(* CoDeSys 2.3.9.62 project: MM000-P9020-00-A.pro *)
(* Author: JvL *)
(* Libraries: ifm_CR0451\ifm_CR0451_Init_V030000.lib 23.10.20 12:28:47, ifm_CR0451\ifm_CR0451_V030002.lib 22.3.17 09:59:30, ifm_RAWCan\ifm_RAWCan_NT_V020004.lib 1.10.19 08:10:40, ifm_CANopen\ifm_CANopen_NT_V020004.lib 1.10.19 08:10:40, ifm_CANopen\ifm_NetVarLib_NT_V020004.lib 1.10.19 08:10:40, ifm_CANopen\3S_CANopenManager.lib 23.10.20 12:28:45, ifm_CANopen\3S_CanDrv.lib 23.10.20 12:28:45, Util.lib 23.10.20 12:25:49, ifm_PDMsmart_util_V010007.lib 23.10.20 12:28:45, Iecsfc.lib 2.6.14 11:37:46, 3S_CANOPENNETVAR.LIB 23.10.20 12:28:45, standard.lib 4.10.05 12:14:46, SysLibVisuBasicDisplay.lib 22.3.17 09:59:30, SysLibTargetVisu.lib 5.4.04 14:31:00, SysLibCallback.lib 26.9.08 18:43:52, ifm_CR0451_callback_visu.lib 23.10.20 12:28:47, SysLibStr.lib 13.6.03 16:49:00 *)

(* PLC configuration (modules and I/O channels)
CR0451 Configuration V03 [Root] node -1, in %IB0 out %QB0
  Configuration [LocalConfiguration] node 0, in %IB0 out %QB0 {IFM_PARAM_WORD_TIME = 10}
  Input/Output [LocalInputOutput] node 1, in %IB0 out %QB0
    Display Keys [LocalKeys] node 0, in %IB0 out %QB0
      KEY_F1 AT %IB0 [ChInputBool] F1 Key
      KEY_F2 AT %IB1 [ChInputBool] F2 Key
      KEY_F3 AT %IB2 [ChInputBool] F3 Key
      KEY_F4 AT %IB3 [ChInputBool] F4 Key
      KEY_UP AT %IB4 [ChInputBool] Up Key
      KEY_DOWN AT %IB5 [ChInputBool] Down Key
      KEY_LEFT AT %IB6 [ChInputBool] Left Key
      KEY_RIGHT AT %IB7 [ChInputBool] Right Key
      KEY_OK AT %IB8 [ChInputBool] Ok Key
    Virtual Raising Keys [VirtualRaisingKeys] node 1, in %IB9 out %QB0
      RT_F1 AT %IB9 [ChInputBool] Rising Edge F1 Key
      RT_F2 AT %IB10 [ChInputBool] Rising Edge F2 Key
      RT_F3 AT %IB11 [ChInputBool] Rising Edge F3 Key
      RT_F4 AT %IB12 [ChInputBool] Rising Edge F4 Key
      RT_UP AT %IB13 [ChInputBool] Rising Edge Up Key
      RT_DOWN AT %IB14 [ChInputBool] Rising Edge Down Key
      RT_LEFT AT %IB15 [ChInputBool] Rising Edge Left Key
      RT_RIGHT AT %IB16 [ChInputBool] Rising Edge Right Key
      RT_OK AT %IB17 [ChInputBool] Rising Edge Ok Key
    Virtual Falling Keys [VirtualFallingKeys] node 2, in %IB18 out %QB0
      FT_F1 AT %IB18 [ChInputBool] Falling Edge F1 Key
      FT_F2 AT %IB19 [ChInputBool] Falling Edge F2 Key
      FT_F3 AT %IB20 [ChInputBool] Falling Edge F3 Key
      FT_F4 AT %IB21 [ChInputBool] Falling Edge F4 Key
      FT_UP AT %IB22 [ChInputBool] Falling Edge Up Key
      FT_DOWN AT %IB23 [ChInputBool] Falling Edge Down Key
      FT_LEFT AT %IB24 [ChInputBool] Falling Edge Left Key
      FT_RIGHT AT %IB25 [ChInputBool] Falling Edge Right Key
      FT_OK AT %IB26 [ChInputBool] Falling Edge Ok Key
    Key Events [KeyEvents] node 3, in %IB27 out %QB0
      KEY_CHANGED AT %IB27 [ChInputBool] Event: Key Changed
      KEY_PRESSED AT %IB28 [ChInputBool] Event: Key is pressed
    System Inputs [LocalSystemInputs] node 4, in %IB29 out %QB0
      SUPPLY_VOLTAGE_VBBS AT %IW15 [ChInputWord] Supply voltage VBBS
      SUPPLY_VOLTAGE_VU AT %IW16 [ChInputWord] Supply voltage VU
      TEMPERATURE AT %IW17 [ChInputInt] Temperature
    Backlight Control [LocalBacklightControl] node 5, in %IB36 out %QB0
      SCREEN_BACKLIGHT_CTRL AT %QB0 [ChOutputByte] Screen Backlight (0 - 100%)
      KEY_BACKLIGHT_CTRL AT %QB1 [ChOutputByte] Key Backlight (0 - 100%)
  CAN Communication [LocalCANCom] node 2, in %IB36 out %QB2
    Interface CAN 1 [CAN_BUS] node 0, in %IB36 out %QB2 {STACK_DWORD_S = 0}
      CANopen Interface [CAN_OPEN] node 0, in %IB36 out %QB2
      J1939 Interface [CAN_J1939] node 1, in %IB36 out %QB2
*)

(* Global variable list: CanOpen implicit Variables *)
VAR_GLOBAL CONSTANT
	MAX_CTRLINDEX : INT := -1;
END_VAR

(* Global variable list: Global_Variables *)
VAR_GLOBAL
	alarm: BOOL;
	editMode: BOOL;
	brakesAlarm: BOOL;
	overloadWarningBlink: BOOL;
	sensorFailureBlink: BOOL;
	overspeedAlarmBlink: BOOL;
	cr0451VersionNo: STRING;
	prefix: STRING;
END_VAR

VAR_GLOBAL RETAIN
	bandLimit: BYTE;
	wcbLimit: BYTE;
END_VAR

(* Global variable list: Networkmanagement implicit Variables CAN *)
VAR_GLOBAL CONSTANT
	USE_NWVARS_CAN : BOOL := TRUE;
	MAX_NetVarItems_CAN	: INT := 23;
	MAX_NetVarPDO_Rx_CAN	: INT := 6;
	MAX_NetVarPDO_Tx_CAN	: INT := 0;
	MAX_NetVarOD_CAN		: INT := 0;
END_VAR
VAR_GLOBAL
	pNetVarItems_CAN		: ARRAY[0..MAX_NetVarItems_CAN] OF NetVarDataItem_CAN;
	pNetVarPDO_Rx_CAN		: ARRAY[0..MAX_NetVarPDO_Rx_CAN] OF NetVarPDO_Rx_CAN;
	pNetVarPDO_Tx_CAN		: ARRAY[0..MAX_NetVarPDO_Tx_CAN] OF NetVarPDO_Tx_CAN;
	pNetVarOD_CAN			: ARRAY[0..MAX_NetVarOD_CAN] OF NetVarOD_CAN;
END_VAR

(* Global variable list: PDM_PLC_COMUNICATION2 *)
VAR_GLOBAL

	(*
	 System variables for basic comunication. CANopen TX/RX PDO1, PDO2, PDO3 and PDO4
	or CANLayer2 TX/RX COB1, COB2, COB3 and COB4
	*)


(************************************From PDM to PLC**********************************************************)

	PRESENT_PAGE:WORD;					(*Preset page number from PDM to PLC*)
	PRESENT_MESSAGE:BYTE;					(*Preset message number from PDM to PLC*)
	PRESENT_MESSAGE_GROUP:BYTE;		(*Preset message group number from PDM to PLC*)
	F_KEYS:BYTE;								(*Funtion keys F1 to F8 from PDM to PLC*)
	C_KEYS:BYTE;								(*Control keys from PDM to PLC*)
	PRESENT_LEDVALUE_MAX:BYTE;			(*Preset LED valus max from PDM to PLC*)
	PRESENT_LEDVALUE_NIGHT:BYTE;		(*Preset LED value night from PDM to PLC*)

	PRESENT_BACKLIGHT:BYTE;				(*Preset backlight value from PDM to PLC*)
	HANDLE:WORD;								(*Handle for input value to PLC*)
	INPUT_VALUE:DWORD;						(*Input value to PLC*)
	LENGHT:BYTE;								(*Length for input value*)

	F_KEYS2:				BYTE;					(*Funtion keys F9 to F16 from PDM to PLC*)
	ToPlcPdo3ReserveByte1:BYTE;					(*Reserve PDO*)
	ToPlcPdo3ReserveByte2:BYTE;					(*Reserve PDO*)
	ToPlcPdo3ReserveByte3:BYTE;					(*Reserve PDO*)
	ToPlcPdo3ReserveByte4:BYTE;					(*Reserve PDO*)
	ToPlcPdo3ReserveByte5:BYTE;					(*Reserve PDO*)
	ToPlcPdo3ReserveByte6:BYTE;					(*Reserve PDO*)
	ToPlcPdo3ReserveByte7:BYTE;					(*Reserve PDO*)

	ToPlcPdo4ReserveByte0:BYTE;					(*Reserve PDO*)
	ToPlcPdo4ReserveByte1:BYTE;					(*Reserve PDO*)
	ToPlcPdo4ReserveByte2:BYTE;					(*Reserve PDO*)
	ToPlcPdo4ReserveByte3:BYTE;					(*Reserve PDO*)
	ToPlcPdo4ReserveByte4:BYTE;					(*Reserve PDO*)
	ToPlcPdo4ReserveByte5:BYTE;					(*Reserve PDO*)
	ToPlcPdo4ReserveByte6:BYTE;					(*Reserve PDO*)
	ToPlcPdo4ReserveByte7:BYTE;					(*Reserve PDO*)

(*^^^^^^^^^^^^^^^^^^^^^^^^^^^^^^^^^^^^^^^^^^^^^^^^^^^^^^^^^^^^^^^^^^^^^^^^^^^^^^^^^^^^^^^^^^^^^^^^^^^^^^^^^^^^^^^^^^^^^^^^^^^^^^^^^^^^^^^^^^*)

(*********************************************From PLC to PDM****************************************************************************)

	DESIRED_PAGE:WORD;						(*Desired page number from PLC to PDM*)
	DESIRED_MESSAGE:BYTE;					(*Desired message number from PLC to PDM*)
	DESIRED_MESSAGE_GROUP:BYTE;		(*Desired message group number from PLC to PDM*)
	LED_F_KEYS:BYTE;							(*LED Funtion keys F1 to F8 from PLC to PDM*)
	LED_C_KEYS:BYTE;							(*LED Control keys from PLC to PDM*)
	DESIRED_LEDVALUE_MAX:BYTE;			(*Desired LED valus max from PLC to PDM*)
	DESIRED_LEDVALUE_NIGHT:BYTE;		(*Desired LED value night from PLC to PDM*)

	DESIRED_BACKLIGHT:BYTE;				(*Desired backlight value from PLC to PDM*)
	HANDLE_BACK:WORD;						(*Handle for input value, write back from PLC*)
	INPUT_VALUE_BACK:DWORD;				(*Input value, write back from PLC*)
	LENGHT_BACK:BYTE;						(*Length for input value, write back from PLC*)

	LED_F_KEYS2		:BYTE;					(*LED Funtion keys F9 to F16 from PLC to PDM*)
	ToPdmPdo3ReserveByte1:BYTE;					(*Reserve PDO*)
	ToPdmPdo3ReserveByte2:BYTE;					(*Reserve PDO*)
	ToPdmPdo3ReserveByte3:BYTE;					(*Reserve PDO*)
	ToPdmPdo3ReserveByte4:BYTE;					(*Reserve PDO*)
	ToPdmPdo3ReserveByte5:BYTE;					(*Reserve PDO*)
	ToPdmPdo3ReserveByte6:BYTE;					(*Reserve PDO*)
	ToPdmPdo3ReserveByte7:BYTE;					(*Reserve PDO*)

	ToPdmPdo4ReserveByte0:BYTE;					(*Reserve PDO*)
	ToPdmPdo4ReserveByte1:BYTE;					(*Reserve PDO*)
	ToPdmPdo4ReserveByte2:BYTE;					(*Reserve PDO*)
	ToPdmPdo4ReserveByte3:BYTE;					(*Reserve PDO*)
	ToPdmPdo4ReserveByte4:BYTE;					(*Reserve PDO*)
	ToPdmPdo4ReserveByte5:BYTE;					(*Reserve PDO*)
	ToPdmPdo4ReserveByte6:BYTE;					(*Reserve PDO*)
	ToPdmPdo4ReserveByte7:BYTE;					(*Reserve PDO*)

(*^^^^^^^^^^^^^^^^^^^^^^^^^^^^^^^^^^^^^^^^^^^^^^^^^^^^^^^^^^^^^^^^^^^^^^^^^^^^^^^^^^^^^^^^^^^^^^^^^^^^^^^^^^^^^^^^^^^^^^^^^^^^^^^^^^^^^^^^^^*)

END_VAR

(* Global variable list: SOFTKEYFIELD *)
VAR_GLOBAL

	(*Variables Input and for text attribute*)
	InputModeDt: BOOL;
	TextColor:DWORD:=16#FFFFFF;
	TextSize:BYTE:=12;

	(*Variables to hide and show the key fields*)
	Hidden_F1:BOOL;
	Hidden_F2:BOOL;
	Hidden_F3:BOOL;
	Hidden_F4:BOOL;
	Hidden_F5:BOOL;
	Hidden_F6:BOOL;
	Hidden_F7:BOOL;
	Hidden_F8:BOOL;
	Hidden_F9:BOOL;
	Hidden_Ctrl:BOOL;
	Hidden_Up:BOOL;
	Hidden_Down:BOOL;
	Hidden_Left:BOOL;
	Hidden_Right:BOOL;
	Hidden_Ok:BOOL;
	Hidden_HeadLine:BOOL;

	(*
	String variables for softkeys.
	With string size 14 it ist possible to show two lines with 6 characters.
	Two character are use for CR/LF Ee.g.ROW_11 $R$NROW_22
	*)
	TXT_F1:STRING[20];
	TXT_F2:STRING[20];
	TXT_F3:STRING[20];
	TXT_F4:STRING[20];
	TXT_F5:STRING[20];
	TXT_F6:STRING[20];
	TXT_F7: STRING[20];
	TXT_F8: STRING[20];
	TXT_F9: STRING[20];
	TXT_Ctrl: STRING[20];
	TXT_HeadLine :STRING[30];

END_VAR

(* Global variable list: SoftKeys2Global *)
VAR_GLOBAL
(*Soft key's as R_TRIG*)
	SoftKey_F1: BOOL;
	SoftKey_F2: BOOL;
	SoftKey_F3: BOOL;
	SoftKey_F4: BOOL;
	SoftKey_F5: BOOL;
	SoftKey_F6: BOOL;
	SoftKey_F7: BOOL;
	SoftKey_F8: BOOL;
	SoftKey_F9: BOOL;
	SoftKey_F10: BOOL;
	SoftKey_Up: BOOL;
	SoftKey_Esc: BOOL;
	SoftKey_Ok: BOOL;
	SoftKey_Left: BOOL;
	SoftKey_Down: BOOL;
	SoftKey_Right: BOOL;
(*Soft key's as switch*)
	SoftKey2_F1: BOOL;
	SoftKey2_F2: BOOL;
	SoftKey2_F3: BOOL;
	SoftKey2_F4: BOOL;
	SoftKey2_F5: BOOL;
	SoftKey2_F6: BOOL;
	SoftKey2_F7: BOOL;
	SoftKey2_F8: BOOL;
	SoftKey2_F9: BOOL;
	SoftKey2_F10: BOOL;
	SoftKey2_Up: BOOL;
	SoftKey2_Esc: BOOL;
	SoftKey2_Ok: BOOL;
	SoftKey2_Left: BOOL;
	SoftKey2_Down: BOOL;
	SoftKey2_Right: BOOL;
	InputMode:BOOL;

END_VAR

(* POU PLC_PRG, FBD *)
PROGRAM PLC_PRG
(*******************************************************************************************************************

			Template for CR0451 V03 - CAN layer 2 (2014)
			--------------------------------------------

	Wir möchten an dieser Stelle ausdrücklich darauf hinweisen, dass die eingestellten Beispiele
	nicht ungeprüft industriell eingesetzt werden dürfen. Das heißt, dass wir für die Funktionalität
	insbesondere an Maschinen und Anlagen keinerlei Garantie übernehmen. Das Beispiel ist
	ausschließlich für Testzwecke bei der Entwicklung neuer Maschinen und Anlagen vorgesehen
	und wurde dafür in Abstimmung mit Ihnen konstruiert und hergestellt. Insoweit handelt es sich
	nicht um ein (Software-) Produkt, das von europäischen Richtlinien erfasst wird. Die Konformität
	mit einschlägigen Richtlinien und Normen zur Erfüllung der gesetzlichen Anforderungen für das
	Inverkehrbringen werden erst mit der Verifizierung und Validierung im Rahmen Ihrer Entwicklung
	festgestellt. Ein Bereitstellen auf dem Markt zur Verwendung durch Endnutzer darf bis zu diesem
	Zeitpunkt nicht stattfinden. 
 
 	We would like to expressly point out that the examples made available must not be used for industrial
	purposes without checking. We assume no guarantee whatsoever for their functionality, particularly
	regarding machines and plants. The example is only intended for testing during the development of
	new machines and plants and has been designed and manufactured for this purpose in coordination
	with you.  Consequently, it is not a (software) product subject to European directives. Compliance with
	relevant directives and standards to meet legal requirements regarding the placing on the market will
	only be determined during the verification and validation in the context of your development. Until then,
	it must not be put onto the market for use by end users.

*******************************************************************************************************************)

VAR

	init_1: BOOL := TRUE;
	CycleTime:DWORD;
	MaxCycleTime:DWORD;
	ResetMax:BOOL;

	Start_time: TIME;


	fbBlink02: BLINK;
END_VAR
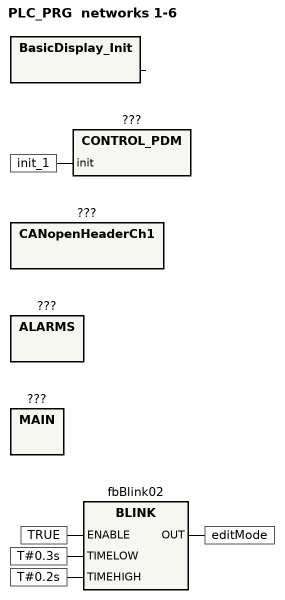
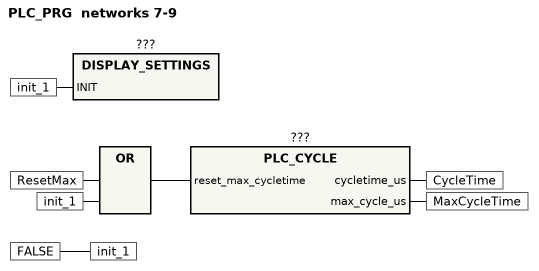
_FBD_ (* Function Block Diagram *)
NETWORK 1
	BasicDisplay_Init()
NETWORK 2
	???:CONTROL_PDM(init: init_1)
NETWORK 3
	???:CANopenHeaderCh1()
NETWORK 4
	???:ALARMS()
NETWORK 5
	???:MAIN()
NETWORK 6
	fbBlink02:BLINK(ENABLE: TRUE, TIMELOW: T#0.3s, TIMEHIGH: T#0.2s) => editMode
NETWORK 7
	???:DISPLAY_SETTINGS(INIT: init_1)
NETWORK 8
	???:PLC_CYCLE(reset_max_cycletime: OR(ResetMax, init_1), max_cycle_us => MaxCycleTime) => CycleTime
NETWORK 9 (* second last line *)
	FALSE => init_1
_END_FBD_
(* the same logic as Structured Text *)
(* Network 1 *)
BasicDisplay_Init();
(* Network 2: see the listing above *)
(* Network 3: see the listing above *)
(* Network 4: see the listing above *)
(* Network 5: see the listing above *)
(* Network 6 *)
fbBlink02(ENABLE := TRUE, TIMELOW := T#0.3s, TIMEHIGH := T#0.2s);
editMode := fbBlink02.OUT;
(* Network 7: see the listing above *)
(* Network 8: see the listing above *)
(* Network 9 *)
init_1 := FALSE;
END_PROGRAM

(* POU CONTROL_CR10xx/CONTROL_PDM, FBD *)
PROGRAM CONTROL_PDM
VAR

	PageIntern: WORD;


	ErrorCom: BOOL;
END_VAR
VAR_INPUT

	init: BOOL;

END_VAR
VAR_OUTPUT
END_VAR
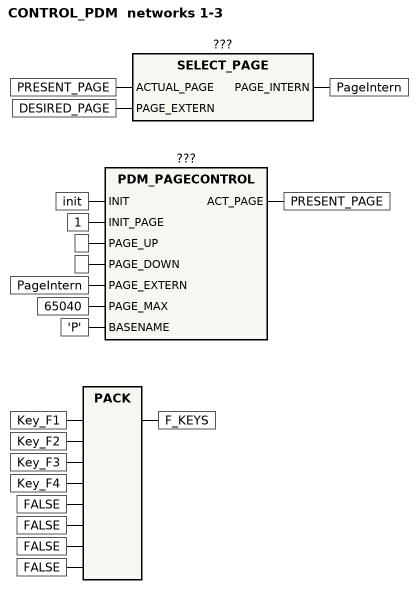
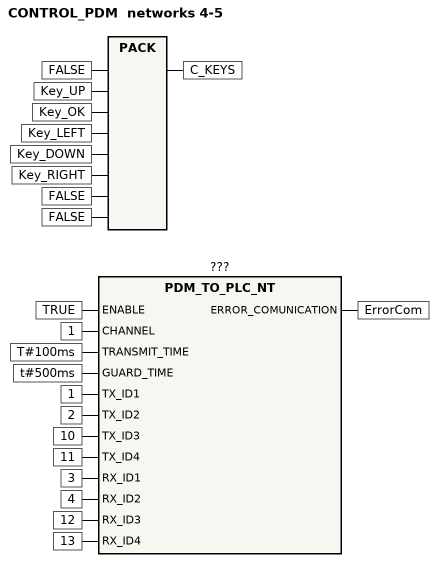
_FBD_ (* Function Block Diagram *)
NETWORK 1 (* This POU must located before PDM_PAGECONTROL, for timing reasons. Include here the program part to change the pages. *)
	???:SELECT_PAGE(ACTUAL_PAGE: PRESENT_PAGE, PAGE_EXTERN: DESIRED_PAGE) => PageIntern
NETWORK 2
	???:PDM_PAGECONTROL(INIT: init, INIT_PAGE: 1, PAGE_UP: , PAGE_DOWN: , PAGE_EXTERN: PageIntern, PAGE_MAX: 65040, BASENAME: 'P') => PRESENT_PAGE
NETWORK 3
	PACK(Key_F1, Key_F2, Key_F3, Key_F4, FALSE, FALSE, FALSE, FALSE) => F_KEYS
NETWORK 4
	PACK(FALSE, Key_UP, Key_OK, Key_LEFT, Key_DOWN, Key_RIGHT, FALSE, FALSE) => C_KEYS
NETWORK 5
	???:PDM_TO_PLC_NT(ENABLE: TRUE, CHANNEL: 1, TRANSMIT_TIME: T#100ms, GUARD_TIME: t#500ms, TX_ID1: 1, TX_ID2: 2, TX_ID3: 10, TX_ID4: 11, RX_ID1: 3, RX_ID2: 4, RX_ID3: 12, RX_ID4: 13) => ErrorCom
_END_FBD_
(* the same logic as Structured Text *)
(* Network 1: see the listing above *)
(* Network 2: see the listing above *)
(* Network 3 *)
F_KEYS := PACK(Key_F1, Key_F2, Key_F3, Key_F4, FALSE, FALSE, FALSE, FALSE);
(* Network 4 *)
C_KEYS := PACK(FALSE, Key_UP, Key_OK, Key_LEFT, Key_DOWN, Key_RIGHT, FALSE, FALSE);
(* Network 5: see the listing above *)
END_PROGRAM

(* POU CONTROL_CR10xx/SELECT_PAGE, ST *)
PROGRAM SELECT_PAGE
(*insert this POU in POU  CONTROL_PDM one line be for PDM_PAGECONTROL!!!!!!!!!!!!!!!!!*)
(*adapt the menue structure for your program in this POU*)
(*10.09.2010 vl FB enhanced by SoftKey2_F1 to SoftKey2_Right as switch*)

VAR_OUTPUT
	PAGE_INTERN: WORD;
END_VAR
VAR_INPUT
	ACTUAL_PAGE: WORD;
	PAGE_EXTERN:WORD;

END_VAR
VAR

	PageExternOld: WORD;

(*Virtual F-keys*)
	VirtualF1: BOOL;
	VirtualF2: BOOL;
	VirtualF3: BOOL;
	VirtualF4: BOOL;
	VirtualF5: BOOL;
	VirtualF6: BOOL;
	VirtualEsc: BOOL;
	VirtualUp: BOOL;
	VirtualOk: BOOL;
	VirtualLeft: BOOL;
	VirtualDown: BOOL;
	VirtualRight: BOOL;

	InputModeStep1: BOOL;
	InputPage: BOOL;
	InputMode:BOOL;
	TOF_InputMode: TOF;
	F_TRIG_InputMode: F_TRIG;

	F5: BOOL;
	InitMenu: BOOL;
	CountMenu: BYTE;
	MenuUp: BOOL;
	MenuDown: BOOL;
	MenuItem: BYTE;
	ItemOk: BOOL;

	Delay: TON;
END_VAR
(*Create virtual keys for menu's*)
	SELECT_MENU(
		Count:=CountMenu,
		Up:= MenuUp,
		Down:=MenuDown,
		MenuItem=>MenuItem );

	VirtualF1:=MenuItem=1 AND Key_Ok;
	VirtualF2:=MenuItem=2 AND Key_Ok;
	VirtualF3:=MenuItem=3 AND Key_Ok;
	VirtualF4:=MenuItem=4 AND Key_Ok;
	VirtualF5:=MenuItem=5 AND Key_Ok;
	VirtualF6:=MenuItem=6 AND Key_Ok;
(*^^^^^^^^^^^^^^^^^^^^^^^^^^^^^^^^^^^^^^^^^^^^^^^^^^^^^^^^^^^^^^^^^^^^^^^^^^^^^^^^^^^^^^^^^^*)

(*Use on following pages the real keys*)
	CASE ACTUAL_PAGE OF
		10:
				VirtualF1:= Key_F1;
				VirtualF2:= Key_F2;
				VirtualF3:= Key_F3;
		12:
				VirtualF1:= Key_F1;
				VirtualF2:= Key_F2;
				VirtualF4:= Key_F4;
		65020:
				VirtualF1:= Key_F1;
				VirtualF2:= Key_F2;
		65030:
				VirtualF1:= Key_F1;

	END_CASE;
(*^^^^^^^^^^^^^^^^^^^^^^^^^^^^^^^^^^^^^^^^^^^^^^^^^^^^^^^^^^^^^^^^^^^^^^^^^^^^^^^^^^^^^^^^^^*)

(*Create soft keys*)
	RT_SOFT_KEYS2(
		KEY_F1:=VirtualF1,
		KEY_F2:=VirtualF2,
		KEY_F3:=VirtualF3,
		KEY_F4:=VirtualF4,
		KEY_F5:=VirtualF5,
		KEY_F6:=VirtualF6,
		KEY_ESC:=Key_F4,
		KEY_UP:=KEY_UP,
		KEY_OK:=KEY_OK,
		KEY_LEFT:=KEY_LEFT,
		KEY_DOWN:=KEY_DOWN,
		KEY_RIGHT:=KEY_RIGHT );
(*^^^^^^^^^^^^^^^^^^^^^^^^^^^^^^^^^^^^^^^^^^^^^^^^^^^^^^^^^^^^^^^^^^^^^^^^^^^^^^^^^^^^^^^^^^*)

(*Set input mode for PDMsmart*)
	IF InputPage AND (SoftKey_LEFT OR SoftKey_RIGHT) THEN
		InputModeStep1:=TRUE;
	END_IF;
	IF SoftKey_ESC THEN
		InputModeStep1:=FALSE;
	END_IF;
	IF InputMode AND (SoftKey_ESC OR SoftKey_OK) THEN
		InputMode:=FALSE;
		InputModeStep1:=FALSE;
	END_IF;
	IF InputModeStep1 AND NOT InputMode AND SoftKey_OK THEN
		InputMode:=TRUE;
	END_IF;

(*^^^^^^^^^^^^^^^^^^^^^^^^^^^^^^^^^^^^^^^^^^^^^^^^^^^^^^^^^^^^^^^^^^^^^^^^^^^^^^^^^^^^^^^*)

(****PAGE from extern****************)
	IF PageExternOld<>PAGE_EXTERN THEN
		PageExternOld:=PAGE_EXTERN;
		PAGE_INTERN:=PAGE_EXTERN;
	END_IF;
(*^^^^^^^^^^^^^^^^^^^^^^^^^^^^^^^^^^^^^^^^^^^^^^^^^^^^^^^^^^^^^^^^*)

	CASE ACTUAL_PAGE OF
(********************Start page*******************************)

		1:	Delay(IN:= NOT(Delay.Q), PT:= T#3s);
			IF Delay.Q THEN
				PAGE_INTERN:= 10;
			END_IF
			InputPage:=FALSE;

			TXT_F1:='';
			TXT_F2:='';
			TXT_F3:='';
			TXT_F4:='';
			TXT_HeadLine:='';
			Hidden_F1:=TRUE;
			Hidden_F2:=TRUE;
			Hidden_F3:=TRUE;
			Hidden_F4:=TRUE;
			Hidden_Up:=TRUE;
			Hidden_Down:=TRUE;
			Hidden_Left:=TRUE;
			Hidden_Right:=TRUE;
			Hidden_Ok:=FALSE;
			Hidden_HeadLine:=FALSE;


(*^^^^^^^^^^^^^^^^^^^^^^^^^^^^^^^^^^^^^^^^^^^^^^^^^^^^^^^^^^^^^*)

(**************************Main page***********************************)
		10:
			Delay(IN:= NOT(Delay.Q), PT:= T#1s);
			IF Delay.Q THEN
				PAGE_INTERN:= 10;
			END_IF
			TXT_F1:='';
			TXT_F2:='';
			TXT_F3:='';
			TXT_F4:='';
			TXT_HeadLine:= '';
			Hidden_F1:=TRUE;
			Hidden_F2:=TRUE;
			Hidden_F3:=TRUE;
			Hidden_F4:=TRUE;
			Hidden_Up:=TRUE;
			Hidden_Down:=TRUE;
			Hidden_Left:=TRUE;
			Hidden_Right:=TRUE;
			Hidden_Ok:=TRUE;
			Hidden_HeadLine:=TRUE;

			IF SoftKey_F1 THEN
				PAGE_INTERN:= 16;
			END_IF
			IF SoftKey_F3 AND sensorFailure = FALSE THEN
				PAGE_INTERN:= 12;
				skylineActive:= TRUE;
			END_IF

			InputPage:=FALSE;

(********************************Input status page********************************************)
		11:
			TXT_F1:='';
			TXT_F2:='';
			TXT_F3:='';
			TXT_F4:= '';
			TXT_HeadLine:= 'INPUT STATUS';
			Hidden_F1:= TRUE;
			Hidden_F2:= TRUE;
			Hidden_F3:= TRUE;
			Hidden_F4:= TRUE;
			Hidden_Up:= TRUE;
			Hidden_Down:= TRUE;
			Hidden_Left:= TRUE;
			Hidden_Right:= TRUE;
			Hidden_Ok:= TRUE;
			Hidden_HeadLine:= FALSE;

			IF SoftKey_ESC THEN
				PAGE_INTERN:=16;
			END_IF;

			InputPage:=FALSE;

(********************************Working mode page********************************************)
		12:
			TXT_F1:='';
			TXT_F2:='';
			TXT_F3:='';
			TXT_F4:='';
			TXT_HeadLine:='';
			Hidden_F1:=TRUE;
			Hidden_F2:=TRUE;
			Hidden_F3:=TRUE;
			Hidden_F4:=TRUE;
			Hidden_Up:=TRUE;
			Hidden_Down:=TRUE;
			Hidden_Left:=TRUE;
			Hidden_Right:=TRUE;
			Hidden_Ok:=TRUE;
			Hidden_HeadLine:=FALSE;

			IF SoftKey_F1 THEN
				PAGE_INTERN:= 16;
			END_IF
			IF SoftKey_F2 THEN
				PAGE_INTERN:= 11;
			END_IF
			IF SoftKey_ESC OR sensorFailure = TRUE THEN
				PAGE_INTERN:= 10;
				skylineActive:= FALSE;
			END_IF;

			InputPage:=FALSE;

(********************************Alarm log page********************************************)
		13:
			TXT_F1:='';
			TXT_F2:='';
			TXT_F3:='';
			TXT_F4:='';
			TXT_HeadLine:='ALARMS LOG';
			Hidden_F1:=TRUE;
			Hidden_F2:=TRUE;
			Hidden_F3:=TRUE;
			Hidden_F4:=TRUE;
			Hidden_Up:=TRUE;
			Hidden_Down:=TRUE;
			Hidden_Left:=TRUE;
			Hidden_Right:=TRUE;
			Hidden_Ok:=TRUE;
			Hidden_HeadLine:=FALSE;

			IF SoftKey_ESC THEN
				PAGE_INTERN:= 16;
			END_IF;

			InputPage:=FALSE;

(********************************Output status page********************************************)
		15:
			TXT_F1:='';
			TXT_F2:='';
			TXT_F3:='';
			TXT_F4:= '';
			TXT_HeadLine:= 'OUTPUT STATUS';
			Hidden_F1:= TRUE;
			Hidden_F2:= TRUE;
			Hidden_F3:= TRUE;
			Hidden_F4:= TRUE;
			Hidden_Up:= TRUE;
			Hidden_Down:= TRUE;
			Hidden_Left:= TRUE;
			Hidden_Right:= TRUE;
			Hidden_Ok:= TRUE;
			Hidden_HeadLine:= FALSE;

			IF SoftKey_ESC THEN
				PAGE_INTERN:=16;
			END_IF

			InputPage:=FALSE;

(********************************Software Version Page***********************************)
		14:
			TXT_F1:='';
			TXT_F2:='';
			TXT_F3:='';
			TXT_F4:= '';
			TXT_HeadLine:= 'SOFTWARE VERSION';
			Hidden_F1:= TRUE;
			Hidden_F2:= TRUE;
			Hidden_F3:= TRUE;
			Hidden_F4:= TRUE;
			Hidden_Up:= TRUE;
			Hidden_Down:= TRUE;
			Hidden_Left:= TRUE;
			Hidden_Right:= TRUE;
			Hidden_Ok:= TRUE;
			Hidden_HeadLine:= FALSE;

			IF SoftKey_ESC THEN
				PAGE_INTERN:=16;
			END_IF

			InputPage:=FALSE;

(********************************Settings page********************************************)
		16:
			TXT_F1:='';
			TXT_F2:='';
			TXT_F3:='';
			TXT_F4:='ESC';
			TXT_HeadLine:='SETTINGS';
			Hidden_F1:=TRUE;
			Hidden_F2:=TRUE;
			Hidden_F3:=TRUE;
			Hidden_F4:=TRUE;
			Hidden_Up:=FALSE;
			Hidden_Down:=FALSE;
			Hidden_Left:=TRUE;
			Hidden_Right:=TRUE;
			Hidden_Ok:=FALSE;
			Hidden_HeadLine:=FALSE;

				CountMenu:=5;
				MenuUp:=SoftKey_Up;
				MenuDown:=SoftKey_Down;

				IF SoftKey_ESC AND NOT InputMode THEN
					IF skylineActive THEN
						PAGE_INTERN:=12;
					ELSE
						PAGE_INTERN:= 10;
					END_IF
				END_IF;
				IF SoftKey_F1 THEN
					PAGE_INTERN:=65000;
				END_IF;
				IF SoftKey_F2 THEN
					PAGE_INTERN:=11;
				END_IF;
				IF SoftKey_F3 THEN
					PAGE_INTERN:=15;
				END_IF;
				IF SoftKey_F4 THEN
					PAGE_INTERN:=13;
				END_IF
				IF SoftKey_F5 THEN
					PAGE_INTERN:= 14;
				END_IF

				InputPage:=FALSE;

(********************************Setpoints page********************************************)
		65000:
			TXT_F1:='';
			TXT_F2:='';
			TXT_F3:='';
			TXT_F4:='ESC';
			TXT_HeadLine:='SETPOINTS';
			Hidden_F1:=TRUE;
			Hidden_F2:=TRUE;
			Hidden_F3:=TRUE;
			Hidden_F4:=TRUE;
			Hidden_Up:=FALSE;
			Hidden_Down:=FALSE;
			Hidden_Left:=FALSE;
			Hidden_Right:=FALSE;
			Hidden_Ok:=FALSE;
			Hidden_HeadLine:=FALSE;

				CountMenu:=2;
				MenuUp:=SoftKey_Up;
				MenuDown:=SoftKey_Down;

				IF SoftKey_ESC AND NOT InputMode THEN
					CountMenu:=1;
					PAGE_INTERN:=16;
				END_IF;
				IF SoftKey_F1 THEN
					PAGE_INTERN:=60013;
				END_IF;
				IF SoftKey_F2 THEN
					PAGE_INTERN:=60014;
				END_IF;

				InputPage:=FALSE;

(********************************Band brake setpoint page********************************************)
		60013:
			TXT_F1:='';
			TXT_F2:='';
			TXT_F3:='';
			TXT_F4:='ESC';
			TXT_HeadLine:='SETPOINTS';
			Hidden_F1:=TRUE;
			Hidden_F2:=TRUE;
			Hidden_F3:=TRUE;
			Hidden_F4:=TRUE;
			Hidden_Up:=FALSE;
			Hidden_Down:=FALSE;
			Hidden_Left:=FALSE;
			Hidden_Right:=FALSE;
			Hidden_Ok:=FALSE;
			Hidden_HeadLine:=FALSE;

			IF SoftKey_Right THEN
				bandLimit:=bandLimit+5;
			END_IF;
			IF SoftKey_Left THEN
				bandLimit:=bandLimit-5;
			END_IF;
			IF bandLimit < 50 THEN
				bandLimit:=50;
			END_IF;
			IF bandLimit > 100 THEN
				bandLimit:=100;
			END_IF

			IF SoftKey_OK AND NOT InputMode THEN
				bandLimitSetpoint:=bandLimit;
				PAGE_INTERN:=65000;
			END_IF;
			InputPage:=FALSE;

(********************************Water cooled brake setpoint page**************************************)
		60014:
			TXT_F1:='';
			TXT_F2:='';
			TXT_F3:='';
			TXT_F4:='ESC';
			TXT_HeadLine:='SETPOINTS';
			Hidden_F1:=TRUE;
			Hidden_F2:=TRUE;
			Hidden_F3:=TRUE;
			Hidden_F4:=TRUE;
			Hidden_Up:=FALSE;
			Hidden_Down:=FALSE;
			Hidden_Left:=FALSE;
			Hidden_Right:=FALSE;
			Hidden_Ok:=FALSE;
			Hidden_HeadLine:=FALSE;

			IF SoftKey_Right THEN
				wcbLimit:=wcbLimit+5;
			END_IF;
			IF SoftKey_Left THEN
				wcbLimit:=wcbLimit-5;
			END_IF;
			IF wcbLimit < 50 THEN
				wcbLimit:=50;
			END_IF;
			IF wcbLimit > 100 THEN
				wcbLimit:=100;
			END_IF

			IF SoftKey_OK THEN
				wcbLimitSetpoint:=wcbLimit;
				PAGE_INTERN:=65000;
			END_IF;
			InputPage:=FALSE;

(*^^^^^^^^^^^^^^^^^^^^^^^^^^^^^^^^^^^^^^^^^^End pages^^^^^^^^^^^^^^^^^^^^^^^^^^^^^^^^^^^^^^^^^^^^*)

	END_CASE;

(*reset variables for change page. Only CR105x by using Input->Tap Variable*)
	VirtualF1:=FALSE;
	VirtualF2:=FALSE;
	VirtualF3:=FALSE;
	VirtualF4:=FALSE;
	VirtualF5:=FALSE;
	VirtualF6:=FALSE;
	VirtualEsc:=FALSE;
	VirtualUp:= FALSE;
	VirtualOk:= FALSE;
	VirtualLeft:= FALSE;
	VirtualDown:= FALSE;
	VirtualRight:= FALSE;
END_PROGRAM

(* POU CONTROL_CR10xx/SELECT_MENU, ST *)
PROGRAM SELECT_MENU
VAR_INPUT
	Count:BYTE;
	Up:BOOL;
	Down:BOOL;
END_VAR
VAR_OUTPUT
	MenuItem:BYTE:=1;

END_VAR
VAR
	R_TRIG_Up: R_TRIG;
	R_TRIG_Down: R_TRIG;
END_VAR
	R_TRIG_Up(CLK:=Up , Q=> );
	R_TRIG_Down(CLK:=Down , Q=> );

	IF R_TRIG_Up.Q THEN
		MenuItem:=MenuItem-1;
	END_IF;

	IF MenuItem>Count THEN
		MenuItem:=1;
	END_IF;

	IF R_TRIG_Down.Q THEN
		MenuItem:=MenuItem+1;
	END_IF;

	IF MenuItem<1 THEN
		MenuItem:=Count;
	END_IF;
END_PROGRAM

(* POU CONTROL_CR10xx/RT_SOFT_KEYS2, ST *)
PROGRAM RT_SOFT_KEYS2
VAR_INPUT
	KEY_F1:BOOL;
	KEY_F2:BOOL;
	KEY_F3:BOOL;
	KEY_F4:BOOL;
	KEY_F5:BOOL;
	KEY_F6:BOOL;
	KEY_F7:BOOL;
	KEY_F8:BOOL;
	KEY_F9:BOOL;
	KEY_F10:BOOL;
	KEY_ESC:BOOL;
	KEY_UP:BOOL;
	KEY_OK:BOOL;
	KEY_LEFT:BOOL;
	KEY_DOWN:BOOL;
	KEY_RIGHT:BOOL;
END_VAR
{library private}
VAR

	R_TRIG_F1: R_TRIG;
	R_TRIG_F2: R_TRIG;
	R_TRIG_F3: R_TRIG;
	R_TRIG_F4: R_TRIG;
	R_TRIG_F5: R_TRIG;
	R_TRIG_F6: R_TRIG;
	R_TRIG_F7: R_TRIG;
	R_TRIG_F8: R_TRIG;
	R_TRIG_F9: R_TRIG;
	R_TRIG_F10: R_TRIG;

	R_TRIG_ESC: R_TRIG;
	R_TRIG_UP: R_TRIG;
	R_TRIG_OK: R_TRIG;
	R_TRIG_LEFT: R_TRIG;
	R_TRIG_DOWN: R_TRIG;
	R_TRIG_RIGHT: R_TRIG;

END_VAR
(*Rising trigs*)
	R_TRIG_F1(CLK:=KEY_F1 , Q=>SoftKey_F1 );
	R_TRIG_F2(CLK:=KEY_F2 , Q=>SoftKey_F2 );
	R_TRIG_F3(CLK:=KEY_F3 , Q=>SoftKey_F3 );
	R_TRIG_F4(CLK:=KEY_F4 , Q=>SoftKey_F4 );
	R_TRIG_F5(CLK:=KEY_F5 , Q=>SoftKey_F5 );
	R_TRIG_F6(CLK:=KEY_F6 , Q=>SoftKey_F6 );
	R_TRIG_F7(CLK:=KEY_F7 , Q=>SoftKey_F7 );
	R_TRIG_F8(CLK:=KEY_F8 , Q=>SoftKey_F8 );
	R_TRIG_F9(CLK:=KEY_F9 , Q=>SoftKey_F9 );
	R_TRIG_F10(CLK:=KEY_F10 , Q=>SoftKey_F10 );

	R_TRIG_ESC(CLK:=KEY_ESC , Q=>SoftKey_Esc );
	R_TRIG_UP(CLK:=KEY_UP , Q=>SoftKey_Up );
	R_TRIG_OK(CLK:=KEY_OK , Q=>SoftKey_Ok );
	R_TRIG_LEFT(CLK:=KEY_LEFT , Q=>SoftKey_Left );
	R_TRIG_DOWN(CLK:=KEY_DOWN , Q=>SoftKey_Down );
	R_TRIG_RIGHT(CLK:=KEY_RIGHT, Q=>SoftKey_Right );

(*Static*)
	SoftKey2_F1:=KEY_F1;
	SoftKey2_F2:=KEY_F2;
	SoftKey2_F3:=KEY_F3;
	SoftKey2_F4:=KEY_F4;
	SoftKey2_F5:=KEY_F5;
	SoftKey2_F6:=KEY_F6;
	SoftKey2_F7:=KEY_F7;
	SoftKey2_F8:=KEY_F8;
	SoftKey2_F9:=KEY_F9;
	SoftKey2_F10:=KEY_F10;
	SoftKey2_Esc:=KEY_ESC;
	SoftKey2_Up:=KEY_UP;
	SoftKey2_Ok:=KEY_OK;
	SoftKey2_Left:=KEY_LEFT;
	SoftKey2_Down:=KEY_DOWN;
	SoftKey2_Right:=KEY_RIGHT;
END_PROGRAM

(* POU CONTROL_CR10xx/PDM_TO_PLC_NT, ST *)
PROGRAM PDM_TO_PLC_NT
VAR_INPUT

	ENABLE: BOOL;
	CHANNEL: BYTE;
	TRANSMIT_TIME:TIME;	(*if transmit time=0, both id's transmit asynchron*)
	GUARD_TIME:TIME;
	TX_ID1: WORD;
	TX_ID2: WORD;
	TX_ID3: WORD;
	TX_ID4: WORD;
	RX_ID1:WORD;
	RX_ID2:WORD;
	RX_ID3:WORD;
	RX_ID4:WORD;


END_VAR
VAR_OUTPUT

	ERROR_COMUNICATION: BOOL;

END_VAR
VAR

	Send1: CAN_TX;
	Send2: CAN_TX;
	Send3: CAN_TX;
	Send4: CAN_TX;
	Rec1: CAN_RX;
	Rec2: CAN_RX;
	Rec3: CAN_RX;
	Rec4: CAN_RX;
	async_send1: BOOL;
	async_send2: BOOL;
	async_send3: BOOL;
	async_send4: BOOL;

	clock: BOOL;
	VarDword:DWORD;
	VarWord:WORD;
	T1: TON;
	one: BOOL;
	rec_ok: BOOL;

	Fl_rec_ok: R_TRIG;
	T_guard_on: TON;
	T_guard_off: TON;
	guard_clock_on: BOOL;
	guard_clock_off: BOOL;


	page_old: WORD;
	message_old: BYTE;
	message_group_old: BYTE;
	led_F_key_old: BYTE;
	led_control_key_old: BYTE;
	led_value_max_old: BYTE;
	led_value_night_old: BYTE;
	BacklightOld:BYTE;
	HandleOld:WORD;
	InputValueOld:DWORD;
	LengthOld:BYTE;



	NoGuarding: BOOL;
	Send2Old: BOOL;
	NoSync: BOOL;

	F_Keys2Old: BYTE;
	ToPlcPdo3ReserveByte1Old: BYTE;
	ToPlcPdo3ReserveByte2Old: BYTE;
	ToPlcPdo3ReserveByte3Old: BYTE;
	ToPlcPdo3ReserveByte4Old: BYTE;
	ToPlcPdo3ReserveByte5Old: BYTE;
	ToPlcPdo3ReserveByte6Old: BYTE;
	ToPlcPdo3ReserveByte7Old: BYTE;
	ToPlcPdo4ReserveByte0Old: BYTE;
	ToPlcPdo4ReserveByte1Old: BYTE;
	ToPlcPdo4ReserveByte2Old: BYTE;
	ToPlcPdo4ReserveByte3Old: BYTE;
	ToPlcPdo4ReserveByte4Old: BYTE;
	ToPlcPdo4ReserveByte5Old: BYTE;
	ToPlcPdo4ReserveByte6Old: BYTE;
	ToPlcPdo4ReserveByte7Old: BYTE;

END_VAR
IF enable THEN
(****************Build a sync for transmit*************************)
	IF GUARD_TIME<T#1ms THEN (*if no transmit time stop sync transmition*)
		NoGuarding:=TRUE;
		ELSE
			NoGuarding:=FALSE;
	END_IF;
	IF transmit_time< T#1ms THEN
		NoSync:=TRUE;
		ELSE
			NoSync:=FALSE;
	END_IF;
	IF transmit_time< T#50ms THEN
		transmit_time:=T#50ms;
	END_IF;
	T1(IN:=NOT T1.Q , PT:=transmit_time );
	clock:= T1.Q;

(*^^^^^^^^^^^^^^^^^^^^^^^^^^^^^^^^^^^^^^^^^^^^^^^^^^^^^^^^^^^^^^^^^^*)
(*************************Build the async for transmit*****************)
	IF page_old<>PRESENT_PAGE THEN
		page_old:=PRESENT_PAGE;
		async_send1:=TRUE;
	END_IF;
	IF message_old<>PRESENT_MESSAGE THEN
		message_old:=PRESENT_MESSAGE;
		async_send1:=TRUE;
	END_IF;
	IF message_group_old<>PRESENT_MESSAGE_GROUP THEN
		message_group_old:=PRESENT_MESSAGE_GROUP;
		async_send1:=TRUE;
	END_IF;
	IF led_F_key_old<>F_KEYS THEN
		led_F_key_old:=F_KEYS;
		async_send1:=TRUE;
	END_IF;
	IF led_control_key_old<>C_KEYS THEN
		led_control_key_old:=C_KEYS;
		async_send1:=TRUE;
	END_IF;
	IF led_value_max_old<>PRESENT_LEDVALUE_MAX THEN
		led_value_max_old:=PRESENT_LEDVALUE_MAX;
		async_send1:=TRUE;
	END_IF;
	IF led_value_night_old<>PRESENT_LEDVALUE_NIGHT THEN
		led_value_night_old:=PRESENT_LEDVALUE_NIGHT;
		async_send1:=TRUE;
	END_IF;
	IF PRESENT_BACKLIGHT>100 THEN
		PRESENT_BACKLIGHT:=100;
	END_IF;
	IF BacklightOld<>PRESENT_BACKLIGHT THEN
		BacklightOld:=PRESENT_BACKLIGHT;
		async_send2:=TRUE;
	END_IF;
	IF NoSync THEN
		IF Send2Old<>Send2.DATA[0].7 THEN
			Send2Old:=Send2.DATA[0].7;
			async_send2:=TRUE;
		END_IF;
	END_IF;
	IF HandleOld<>HANDLE THEN
		HandleOld:=HANDLE;
		async_send2:=TRUE;
	END_IF;
	IF InputValueOld<>INPUT_VALUE THEN
		InputValueOld:=INPUT_VALUE;
		async_send2:=TRUE;
	END_IF;
	IF LengthOld<>LENGHT THEN
		LengthOld:=LENGHT;
		async_send2:=TRUE;
	END_IF;
	IF F_Keys2Old<>F_KEYS2 THEN
		F_Keys2Old:=F_KEYS2;
		async_send3:=TRUE;
	END_IF;
	IF ToPlcPdo3ReserveByte1Old<>ToPlcPdo3ReserveByte1 THEN
		ToPlcPdo3ReserveByte1Old:=ToPlcPdo3ReserveByte1;
		async_send3:=TRUE;
	END_IF;
	IF ToPlcPdo3ReserveByte2Old<>ToPlcPdo3ReserveByte2 THEN
		ToPlcPdo3ReserveByte2Old:=ToPlcPdo3ReserveByte2;
		async_send3:=TRUE;
	END_IF;
	IF ToPlcPdo3ReserveByte3Old<>ToPlcPdo3ReserveByte3 THEN
		ToPlcPdo3ReserveByte3Old:=ToPlcPdo3ReserveByte3;
		async_send3:=TRUE;
	END_IF;
	IF ToPlcPdo3ReserveByte4Old<>ToPlcPdo3ReserveByte4 THEN
		ToPlcPdo3ReserveByte4Old:=ToPlcPdo3ReserveByte4;
		async_send3:=TRUE;
	END_IF;
	IF ToPlcPdo3ReserveByte5Old<>ToPlcPdo3ReserveByte5 THEN
		ToPlcPdo3ReserveByte5Old:=ToPlcPdo3ReserveByte5;
		async_send3:=TRUE;
	END_IF;
	IF ToPlcPdo3ReserveByte6Old<>ToPlcPdo3ReserveByte6 THEN
		ToPlcPdo3ReserveByte6Old:=ToPlcPdo3ReserveByte6;
		async_send3:=TRUE;
	END_IF;
	IF ToPlcPdo3ReserveByte7Old<>ToPlcPdo3ReserveByte7 THEN
		ToPlcPdo3ReserveByte7Old:=ToPlcPdo3ReserveByte7;
		async_send3:=TRUE;
	END_IF;
	IF ToPlcPdo4ReserveByte0Old<>ToPlcPdo4ReserveByte0 THEN
		ToPlcPdo4ReserveByte0Old:=ToPlcPdo4ReserveByte0;
		async_send4:=TRUE;
	END_IF;
	IF ToPlcPdo4ReserveByte1Old<>ToPlcPdo4ReserveByte1 THEN
		ToPlcPdo4ReserveByte1Old:=ToPlcPdo4ReserveByte1;
		async_send4:=TRUE;
	END_IF;
	IF ToPlcPdo4ReserveByte2Old<>ToPlcPdo4ReserveByte2 THEN
		ToPlcPdo4ReserveByte2Old:=ToPlcPdo4ReserveByte2;
		async_send4:=TRUE;
	END_IF;
	IF ToPlcPdo4ReserveByte3Old<>ToPlcPdo4ReserveByte3 THEN
		ToPlcPdo4ReserveByte3Old:=ToPlcPdo4ReserveByte3;
		async_send4:=TRUE;
	END_IF;
	IF ToPlcPdo4ReserveByte4Old<>ToPlcPdo4ReserveByte4 THEN
		ToPlcPdo4ReserveByte4Old:=ToPlcPdo4ReserveByte4;
		async_send4:=TRUE;
	END_IF;
	IF ToPlcPdo4ReserveByte5Old<>ToPlcPdo4ReserveByte5 THEN
		ToPlcPdo4ReserveByte5Old:=ToPlcPdo4ReserveByte5;
		async_send4:=TRUE;
	END_IF;
	IF ToPlcPdo4ReserveByte6Old<>ToPlcPdo4ReserveByte6 THEN
		ToPlcPdo4ReserveByte6Old:=ToPlcPdo4ReserveByte6;
		async_send4:=TRUE;
	END_IF;
	IF ToPlcPdo4ReserveByte7Old<>ToPlcPdo4ReserveByte7 THEN
		ToPlcPdo4ReserveByte7Old:=ToPlcPdo4ReserveByte7;
		async_send4:=TRUE;
	END_IF;



(*^^^^^^^^^^^^^^^^^^^^^^^^^^^^^^^^^^^^^^^^^^^^^^^^^^^^^^^^^^^^^^^^^^*)

(************Build the guarding toggle and send it with backlight*****************************)

	IF clock AND (NOT NoSync OR NOT NoGuarding) THEN
		one := NOT one;
	END_IF;

	Send2.DATA[0]:=PRESENT_BACKLIGHT;

	IF one THEN
		Send2.DATA[0].7:= TRUE;
		ELSE
			Send2.DATA[0].7:=FALSE;
	END_IF;
(*^^^^^^^^^^^^^^^^^^^^^^^^^^^^^^^^^^^^^^^^^^^^^^^^^^^^^^^^^^^^^^^^^^*)

(********************copy data to transmit array*********************)

	Send1.DATA[0] := WORD_TO_BYTE(PRESENT_PAGE);
	VarWord := SHR(PRESENT_PAGE,8);
	Send1.DATA[1] := WORD_TO_BYTE(VarWord);
	Send1.DATA[2] := PRESENT_MESSAGE;
	Send1.DATA[3] := PRESENT_MESSAGE_GROUP;
	Send1.DATA[4] := F_KEYS;
	Send1.DATA[5] := C_KEYS;
	Send1.DATA[6] := PRESENT_LEDVALUE_MAX;
	Send1.DATA[7] := PRESENT_LEDVALUE_NIGHT;

	IF LENGHT<1 THEN
		LENGHT:=1;
	END_IF;
	IF LENGHT=3 OR LENGHT>4 THEN
		LENGHT:=4;
	END_IF;

	Send2.DATA[7]:=LENGHT;

	Send2.DATA[1] := WORD_TO_BYTE(HANDLE);
	VarWord := SHR(HANDLE,8);
	Send2.DATA[2] := WORD_TO_BYTE(VarWord);


	CASE LENGHT OF

		1:	Send2.DATA[3]:=DWORD_TO_BYTE(INPUT_VALUE);
			Send2.DATA[4]:=0;
			Send2.DATA[5]:=0;
			Send2.DATA[6]:=0;

		2:	VarDword:=ROL(INPUT_VALUE,32);
			Send2.DATA[3]:=DWORD_TO_BYTE(VarDword);
			VarDword:=ROL(INPUT_VALUE,24);
			Send2.DATA[4]:=DWORD_TO_BYTE(VarDword);
			VarDword:=ROL(INPUT_VALUE,16);
			Send2.DATA[5]:=0;
			Send2.DATA[6]:=0;

		4:	VarDword:=ROL(INPUT_VALUE,32);
			Send2.DATA[3]:=DWORD_TO_BYTE(VarDword);
			VarDword:=ROL(INPUT_VALUE,24);
			Send2.DATA[4]:=DWORD_TO_BYTE(VarDword);
			VarDword:=ROL(INPUT_VALUE,16);
			Send2.DATA[5]:=DWORD_TO_BYTE(VarDword);
			VarDword:=ROL(INPUT_VALUE,8);
			Send2.DATA[6]:=DWORD_TO_BYTE(VarDword);

	END_CASE;

	Send3.DATA[0] := F_KEYS2;
	Send3.DATA[1] := ToPlcPdo3ReserveByte1;
	Send3.DATA[2] := ToPlcPdo3ReserveByte2;
	Send3.DATA[3] := ToPlcPdo3ReserveByte3;
	Send3.DATA[4] := ToPlcPdo3ReserveByte4;
	Send3.DATA[5] := ToPlcPdo3ReserveByte5;
	Send3.DATA[6] := ToPlcPdo3ReserveByte6;
	Send3.DATA[7] := ToPlcPdo3ReserveByte7;

	Send4.DATA[0] := ToPlcPdo4ReserveByte0;
	Send4.DATA[1] := ToPlcPdo4ReserveByte1;
	Send4.DATA[2] := ToPlcPdo4ReserveByte2;
	Send4.DATA[3] := ToPlcPdo4ReserveByte3;
	Send4.DATA[4] := ToPlcPdo4ReserveByte4;
	Send4.DATA[5] := ToPlcPdo4ReserveByte5;
	Send4.DATA[6] := ToPlcPdo4ReserveByte6;
	Send4.DATA[7] := ToPlcPdo4ReserveByte7;


(*^^^^^^^^^^^^^^^^^^^^^^^^^^^^^^^^^^^^^^^^^^^^^^^^^^^^^^^^^^^^^^^^^^^^^^^^^^^^^^^^^^^^*)

(**************send data************************)
	Send1(
	ENABLE:=(clock AND NOT NoSync) OR async_send1 ,
	CHANNEL:=CHANNEL ,
	ID:=Tx_id1 ,
	DATA:= ,
	RESULT=> );

	Send2(
	ENABLE:=(clock AND NOT NoSync) OR async_send2 ,
	CHANNEL:=CHANNEL ,
	ID:=Tx_id2 ,
	DATA:= ,
	RESULT=> );

	Send3(
	ENABLE:=(clock AND NOT NoSync) OR async_send3 ,
	CHANNEL:=CHANNEL ,
	ID:=Tx_id3 ,
	DATA:= ,
	RESULT=> );

	Send4(
	ENABLE:=(clock AND NOT NoSync) OR async_send4 ,
	CHANNEL:=CHANNEL ,
	ID:=Tx_id4 ,
	DATA:= ,
	RESULT=> );

	async_send1:=FALSE;
	async_send2:=FALSE;
	async_send3:=FALSE;
	async_send4:=FALSE;


(*^^^^^^^^^^^^^^^^^^^^^^^^^^^^^^^^^^^^^^^^^^^^^^^^^^^^^^^^^^^^^^^^^^^^^^^^^^^^^^^^^^^^*)

(**************receive data************************)

	Rec1(
	ENABLE:=TRUE ,
	CHANNEL:=CHANNEL ,
	ID:=rx_id1 ,
	DATA=> ,
	RESULT=> );

	Rec2(
	ENABLE:=TRUE ,
	CHANNEL:=CHANNEL ,
	ID:=rx_id2 ,
	DATA=> ,
	RESULT=> );

	Rec3(
	ENABLE:=TRUE ,
	CHANNEL:=CHANNEL ,
	ID:=rx_id3 ,
	DATA=> ,
	RESULT=> );

	Rec4(
	ENABLE:=TRUE ,
	CHANNEL:=CHANNEL ,
	ID:=rx_id4 ,
	DATA=> ,
	RESULT=> );

	(**************************check guarding**********************************)
	Fl_rec_ok(CLK:=Rec2.DATA[0].7 , Q=>rec_ok );

	T_guard_on(IN:=rec_ok , PT:=guard_time , Q=>guard_clock_on);
	T_guard_off(IN:=NOT rec_ok , PT:=guard_time , Q=>guard_clock_off);


	IF NOT NoGuarding AND (guard_clock_on OR guard_clock_off) THEN
		error_comunication := TRUE;
		ELSE
			error_comunication := FALSE;
	END_IF;
	(*^^^^^^^^^^^^^^^^^^^^^^^^^^^^^^^^^^^^^^^^^^^^^^^^^^^^^^^^^^^^^^^^^^^^^^^^^^^^*)

	(***********************copy reveived data***********************************)
	IF Rec1.RESULT=1 THEN
		DESIRED_PAGE := Rec1.DATA[1];
		DESIRED_PAGE := SHL(DESIRED_PAGE,8) OR Rec1.DATA[0];
		DESIRED_MESSAGE := Rec1.DATA[2];
		DESIRED_MESSAGE_GROUP := Rec1.DATA[3];
		LED_F_KEYS := Rec1.DATA[4];
		LED_C_KEYS := Rec1.DATA[5];
		DESIRED_LEDVALUE_MAX := Rec1.DATA[6];
		DESIRED_LEDVALUE_NIGHT := Rec1.DATA[7];
	END_IF;

	IF Rec2.RESULT=1 THEN
		DESIRED_BACKLIGHT:= 16#7F AND Rec2.DATA[0];
		HANDLE_BACK:= BYTE_TO_WORD(Rec2.DATA[2]);
		HANDLE_BACK:=SHL(HANDLE_BACK,8);
		HANDLE_BACK:=HANDLE_BACK OR Rec2.DATA[1];
		LENGHT_BACK:= Rec2.DATA[7];

		IF LENGHT_BACK<1 THEN
			LENGHT_BACK:=1;
		END_IF;
		IF LENGHT_BACK=3 OR LENGHT_BACK>4 THEN
			LENGHT_BACK:=4;
		END_IF;

		CASE LENGHT_BACK OF

			1:	INPUT_VALUE_BACK:=Rec2.DATA[3];

			2:	INPUT_VALUE_BACK:=Rec2.DATA[4];
			INPUT_VALUE_BACK:=SHL(INPUT_VALUE_BACK,8) OR Rec2.DATA[3];

			4:	INPUT_VALUE_BACK:=Rec2.DATA[6];
			INPUT_VALUE_BACK:=SHL(INPUT_VALUE_BACK,8) OR Rec2.DATA[5];
			INPUT_VALUE_BACK:=SHL(INPUT_VALUE_BACK,8) OR Rec2.DATA[4];
			INPUT_VALUE_BACK:=SHL(INPUT_VALUE_BACK,8) OR Rec2.DATA[3];

		END_CASE;
	END_IF;

	IF Rec3.RESULT=1 THEN
		LED_F_KEYS2:=Rec3.DATA[0];
		ToPdmPdo3ReserveByte1:=Rec3.DATA[1];
		ToPdmPdo3ReserveByte2:=Rec3.DATA[2];
		ToPdmPdo3ReserveByte3:=Rec3.DATA[3];
		ToPdmPdo3ReserveByte4:=Rec3.DATA[4];
		ToPdmPdo3ReserveByte5:=Rec3.DATA[5];
		ToPdmPdo3ReserveByte6:=Rec3.DATA[6];
		ToPdmPdo3ReserveByte7:=Rec3.DATA[7];
	END_IF;

	IF Rec4.RESULT=1 THEN
		ToPdmPdo4ReserveByte0:=Rec4.DATA[0];
		ToPdmPdo4ReserveByte1:=Rec4.DATA[1];
		ToPdmPdo4ReserveByte2:=Rec4.DATA[2];
		ToPdmPdo4ReserveByte3:=Rec4.DATA[3];
		ToPdmPdo4ReserveByte4:=Rec4.DATA[4];
		ToPdmPdo4ReserveByte5:=Rec4.DATA[5];
		ToPdmPdo4ReserveByte6:=Rec4.DATA[6];
		ToPdmPdo4ReserveByte7:=Rec4.DATA[7];
	END_IF;

	(*^^^^^^^^^^^^^^^^^^^^^^^^^^^^^^^^^^^^^^^^^^^^^^^^^^^^^^^^^^^^^^^^^^^^^^^^^^^^*)

(*^^^^^^^^^^^^^^^^^^^^^^^^^^^^^^^^^^^^^^^^^^^^^^^^^^^^^^^^^^^^^^^^^^^^^^^^^^^^^^^^^^^^^^^^^^^^^^^^^^^^^^^^^^^^^^^^^^^^^^^^^^^^^^^^^^^^^^^^^^^^*)
END_IF;
END_PROGRAM

(* POU CANopenCh1/CANopenHeaderCh1, FBD *)
PROGRAM CANopenHeaderCh1
VAR

	(*Set CANopen state*)
	SetCanOpenState: CANOPEN_SETSTATE;
	SetState:BOOL:=TRUE;

	(*Handling CANopen status*)
	HandlingCANopen: CANopen_HANDLING_ST;
	SlaveNodeId: BYTE;
	Baudrate: DWORD;
	MasterState: BYTE;
	GuardError: BOOL;
	ErrorNodeList: ARRAY[0..MAXGUARDERR] OF BYTE;
	CanState: BYTE;
	Nodestate: BYTE;
	LastNodeState: BYTE;

	(*Emergency handling*)
	CanEmcy: CAN_EMCY;
	RestEmcyList: BOOL;
	EMCY_MSG_Count: DWORD; (* No of EMCY messages  Leaving errors are count too *)
	EmcyStruct: ARRAY[0..10] OF tT_EMCY;

	(*Handling CAN status*)
	StatusCan: CAN_Status_and_Errors;
	ResetCanFlags: BOOL;
	BusLoad: BYTE;
	BusOff: BOOL;
	RxOverflow: BOOL;
	RxWarning: BOOL;
	TxOverflow: BOOL;
	TxWarning: BOOL;

	EnableCANopen: CANOPEN_ENABLE;
END_VAR
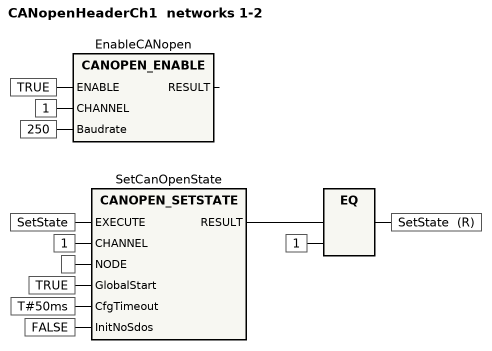
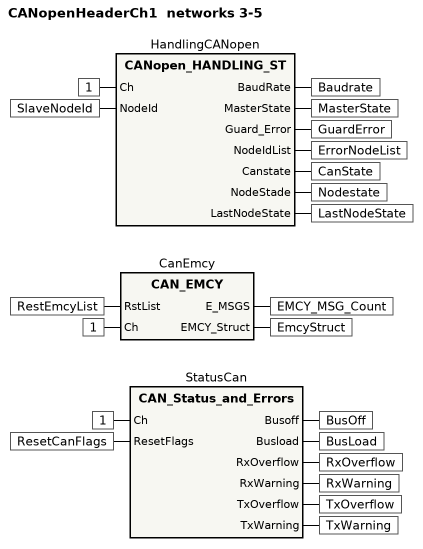
_FBD_ (* Function Block Diagram *)
NETWORK 1 (* Basic functions for the CANopen functionality *)
	EnableCANopen:CANOPEN_ENABLE(ENABLE: TRUE, CHANNEL: 1, Baudrate: 250)
NETWORK 2 (* Set CANopen status *)
	EQ(SetCanOpenState:CANOPEN_SETSTATE(EXECUTE: SetState, CHANNEL: 1, NODE: , GlobalStart: TRUE, CfgTimeout: T#50ms, InitNoSdos: FALSE), 1) => R SetState
NETWORK 3 (* CANopen Master and heartbeat handling *)
	HandlingCANopen:CANopen_HANDLING_ST(Ch: 1, NodeId: SlaveNodeId, MasterState => MasterState, Guard_Error => GuardError, NodeIdList => ErrorNodeList, Canstate => CanState, NodeStade => Nodestate, LastNodeState => LastNodeState) => Baudrate
NETWORK 4 (* CANopen Emergency Handling for 11 emergency messages *)
	CanEmcy:CAN_EMCY(RstList: RestEmcyList, Ch: 1, EMCY_Struct => EmcyStruct) => EMCY_MSG_Count
NETWORK 5 (* Get the CAN Status and CAN Errors *)
	StatusCan:CAN_Status_and_Errors(Ch: 1, ResetFlags: ResetCanFlags, Busload => BusLoad, RxOverflow => RxOverflow, RxWarning => RxWarning, TxOverflow => TxOverflow, TxWarning => TxWarning) => BusOff
_END_FBD_
(* the same logic as Structured Text *)
(* Network 1 *)
EnableCANopen(ENABLE := TRUE, CHANNEL := 1, Baudrate := 250);
(* Network 2: see the listing above *)
(* Network 3 *)
HandlingCANopen(Ch := 1, NodeId := SlaveNodeId);
MasterState := HandlingCANopen.MasterState;
GuardError := HandlingCANopen.Guard_Error;
ErrorNodeList := HandlingCANopen.NodeIdList;
CanState := HandlingCANopen.Canstate;
Nodestate := HandlingCANopen.NodeStade;
LastNodeState := HandlingCANopen.LastNodeState;
Baudrate := HandlingCANopen.BaudRate;
(* Network 4 *)
CanEmcy(RstList := RestEmcyList, Ch := 1);
EmcyStruct := CanEmcy.EMCY_Struct;
EMCY_MSG_Count := CanEmcy.E_MSGS;
(* Network 5 *)
StatusCan(Ch := 1, ResetFlags := ResetCanFlags);
BusLoad := StatusCan.Busload;
RxOverflow := StatusCan.RxOverflow;
RxWarning := StatusCan.RxWarning;
TxOverflow := StatusCan.TxOverflow;
TxWarning := StatusCan.TxWarning;
BusOff := StatusCan.Busoff;
END_PROGRAM

(* POU CANopenCh1/CANopen_HANDLING_ST, ST *)
FUNCTION_BLOCK CANopen_HANDLING_ST
(* CANopen Master and heartbeat handling *)
VAR
	CANOPEN_GETSTATE_: CANOPEN_GETSTATE;
	Execute_Getstate: BOOL := TRUE;
	CANOPEN_GETGUARDHBERRLIST_: CANOPEN_GETGUARDHBERRLIST;
	Execute_Guardlst: BOOL := TRUE;
	ResetErrorList: BOOL;
	PlcNodeId: BYTE;
END_VAR
VAR_INPUT
	Ch: BYTE;
	NodeId: BYTE;
END_VAR
VAR_OUTPUT
	BaudRate: DWORD;
	MasterState: BYTE;
	Guard_Error: BOOL;
	NodeIdList: ARRAY[0..MAXGUARDERR] OF BYTE;
	Canstate: BYTE;
	NodeStade: BYTE;
	LastNodeState: BYTE;
END_VAR
(* ^^^^ Get the current state of the CANopen master ^^^^ *)
CANOPEN_GETSTATE_(
	EXECUTE:=Execute_Getstate ,
	CHANNEL:=Ch ,
	NODE:=NodeId ,
	MASTERSTATE=>MasterState ,
	PLCNODEID=>PlcNodeId ,
	PLCBAUDRATE=>BaudRate ,
	PLCVERSION=>,
	CANSTATE=>Canstate ,
	NODESTATE=>NodeStade ,
	LASTNODESTATE=>LastNodeState ,
	RESULT=> );

(* Values are valid now, function call can be stopped *)
IF CANOPEN_GETSTATE_.RESULT= 1 THEN
	Execute_Getstate:=FALSE;
END_IF

(* Function is passive, execute again *)
IF CANOPEN_GETSTATE_.RESULT= 0 THEN
	Execute_Getstate:=TRUE;
END_IF

(* ^^^^^ Get heartbeaterror or nodeguarding error ^^^^ *)
CANOPEN_GETGUARDHBERRLIST_(
	EXECUTE:=Execute_Guardlst ,
	CHANNEL:=Ch ,
	ResetList:=ResetErrorList ,
	N_NODES=>,
	NODEID=>NodeIdList ,
	RESULT=> );

(* Values are valid now, function call can be stopped *)
IF CANOPEN_GETGUARDHBERRLIST_.RESULT= 1 THEN
		Execute_Guardlst:= FALSE;
END_IF

(* Function is passive, execute again *)
IF CANOPEN_GETGUARDHBERRLIST_.RESULT= 0 THEN
		Execute_Guardlst:= TRUE;
END_IF

(* An heartbeaterror has been appeared *)
IF CANOPEN_GETGUARDHBERRLIST_.N_NODES >0 THEN
	Guard_Error:=TRUE;
ELSE
	Guard_Error:=FALSE;
END_IF;
END_FUNCTION_BLOCK

(* POU CANopenCh1/CAN_EMCY, FBD *)
FUNCTION_BLOCK CAN_EMCY
VAR_INPUT
	RstList: BOOL;
	Ch: BYTE;
END_VAR
VAR_OUTPUT
	E_MSGS: DWORD;
	EMCY_Struct: ARRAY[0..10] OF tT_EMCY;
END_VAR
VAR
	CANOPEN_GETEMCYMESSAGES_: CANOPEN_GETEMCYMESSAGES;
	Get_EMCY_MSG: BOOL := TRUE;
END_VAR
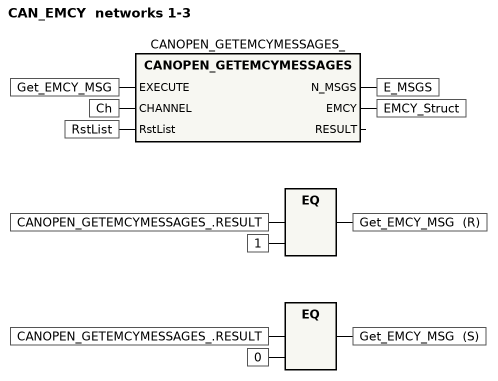
_FBD_ (* Function Block Diagram *)
NETWORK 1
	CANOPEN_GETEMCYMESSAGES_:CANOPEN_GETEMCYMESSAGES(EXECUTE: Get_EMCY_MSG, CHANNEL: Ch, RstList: RstList, EMCY => EMCY_Struct) => E_MSGS
NETWORK 2
	EQ(CANOPEN_GETEMCYMESSAGES_.RESULT, 1) => R Get_EMCY_MSG
NETWORK 3
	EQ(CANOPEN_GETEMCYMESSAGES_.RESULT, 0) => S Get_EMCY_MSG
_END_FBD_
(* the same logic as Structured Text *)
(* Network 1 *)
CANOPEN_GETEMCYMESSAGES_(EXECUTE := Get_EMCY_MSG, CHANNEL := Ch, RstList := RstList);
EMCY_Struct := CANOPEN_GETEMCYMESSAGES_.EMCY;
E_MSGS := CANOPEN_GETEMCYMESSAGES_.N_MSGS;
(* Network 2 *)
IF CANOPEN_GETEMCYMESSAGES_.RESULT = 1 THEN Get_EMCY_MSG := FALSE; END_IF;
(* Network 3 *)
IF CANOPEN_GETEMCYMESSAGES_.RESULT = 0 THEN Get_EMCY_MSG := TRUE; END_IF;
END_FUNCTION_BLOCK

(* POU CANopenCh1/CAN_Status_and_Errors, FBD *)
FUNCTION_BLOCK CAN_Status_and_Errors
(* Get the CAN Status and CAN Errors *)
VAR

	CanStatus:CAN_STATUS;
	GETBUFFERFLAGS: CANOPEN_GETBUFFERFLAGS;

	ExecuteBufferFlags: BOOL:=TRUE;

END_VAR
VAR_INPUT
	Ch: BYTE;

	ResetFlags: BOOL;
END_VAR
VAR_OUTPUT
	Busoff: BOOL;
	Busload: BYTE;
	RxOverflow: BOOL;
	RxWarning: BOOL;
	TxOverflow: BOOL;
	TxWarning: BOOL;
END_VAR
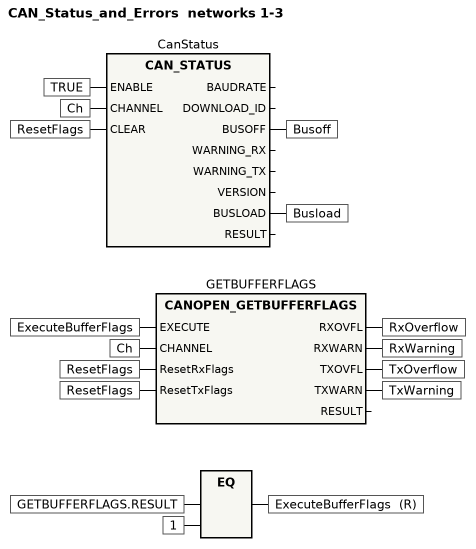
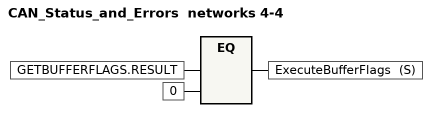
_FBD_ (* Function Block Diagram *)
NETWORK 1 (* Get the CAN Status *)
	CanStatus:CAN_STATUS(ENABLE: TRUE, CHANNEL: Ch, CLEAR: ResetFlags, BUSOFF => Busoff, BUSLOAD => Busload)
NETWORK 2 (* Get Buffer warnings / Reset Buffer Warning *)
	GETBUFFERFLAGS:CANOPEN_GETBUFFERFLAGS(EXECUTE: ExecuteBufferFlags, CHANNEL: Ch, ResetRxFlags: ResetFlags, ResetTxFlags: ResetFlags, RXWARN => RxWarning, TXOVFL => TxOverflow, TXWARN => TxWarning) => RxOverflow
NETWORK 3
	EQ(GETBUFFERFLAGS.RESULT, 1) => R ExecuteBufferFlags
NETWORK 4
	EQ(GETBUFFERFLAGS.RESULT, 0) => S ExecuteBufferFlags
_END_FBD_
(* the same logic as Structured Text *)
(* Network 1: Get the CAN Status *)
CanStatus(ENABLE := TRUE, CHANNEL := Ch, CLEAR := ResetFlags);
Busoff := CanStatus.BUSOFF;
Busload := CanStatus.BUSLOAD;
(* Network 2: Get Buffer warnings / Reset Buffer Warning *)
GETBUFFERFLAGS(EXECUTE := ExecuteBufferFlags, CHANNEL := Ch, ResetRxFlags := ResetFlags, ResetTxFlags := ResetFlags);
RxWarning := GETBUFFERFLAGS.RXWARN;
TxOverflow := GETBUFFERFLAGS.TXOVFL;
TxWarning := GETBUFFERFLAGS.TXWARN;
RxOverflow := GETBUFFERFLAGS.RXOVFL;
(* Network 3 *)
IF GETBUFFERFLAGS.RESULT = 1 THEN ExecuteBufferFlags := FALSE; END_IF;
(* Network 4 *)
IF GETBUFFERFLAGS.RESULT = 0 THEN ExecuteBufferFlags := TRUE; END_IF;
END_FUNCTION_BLOCK

(* POU CONTROL_CR10xx/ALARMS, FBD *)
PROGRAM ALARMS
VAR
	fbBlink01: BLINK;
	fbBlink02: BLINK;
	fbBlink03: BLINK;
	fbBlink04: BLINK;
	fbBlink05: BLINK;
END_VAR
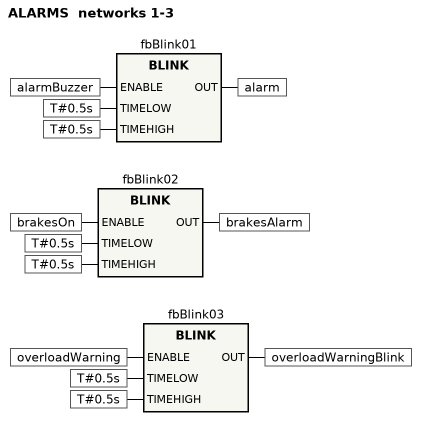
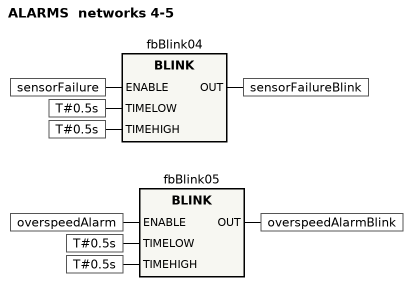
_FBD_ (* Function Block Diagram *)
NETWORK 1
	fbBlink01:BLINK(ENABLE: alarmBuzzer, TIMELOW: T#0.5s, TIMEHIGH: T#0.5s) => alarm
NETWORK 2
	fbBlink02:BLINK(ENABLE: brakesOn, TIMELOW: T#0.5s, TIMEHIGH: T#0.5s) => brakesAlarm
NETWORK 3
	fbBlink03:BLINK(ENABLE: overloadWarning, TIMELOW: T#0.5s, TIMEHIGH: T#0.5s) => overloadWarningBlink
NETWORK 4
	fbBlink04:BLINK(ENABLE: sensorFailure, TIMELOW: T#0.5s, TIMEHIGH: T#0.5s) => sensorFailureBlink
NETWORK 5
	fbBlink05:BLINK(ENABLE: overspeedAlarm, TIMELOW: T#0.5s, TIMEHIGH: T#0.5s) => overspeedAlarmBlink
_END_FBD_
(* the same logic as Structured Text *)
(* Network 1 *)
fbBlink01(ENABLE := alarmBuzzer, TIMELOW := T#0.5s, TIMEHIGH := T#0.5s);
alarm := fbBlink01.OUT;
(* Network 2 *)
fbBlink02(ENABLE := brakesOn, TIMELOW := T#0.5s, TIMEHIGH := T#0.5s);
brakesAlarm := fbBlink02.OUT;
(* Network 3 *)
fbBlink03(ENABLE := overloadWarning, TIMELOW := T#0.5s, TIMEHIGH := T#0.5s);
overloadWarningBlink := fbBlink03.OUT;
(* Network 4 *)
fbBlink04(ENABLE := sensorFailure, TIMELOW := T#0.5s, TIMEHIGH := T#0.5s);
sensorFailureBlink := fbBlink04.OUT;
(* Network 5 *)
fbBlink05(ENABLE := overspeedAlarm, TIMELOW := T#0.5s, TIMEHIGH := T#0.5s);
overspeedAlarmBlink := fbBlink05.OUT;
END_PROGRAM

(* POU MAIN, ST *)
PROGRAM MAIN
VAR
END_VAR
cr0451VersionNo := '020-00-A';
prefix := 'MM000-P9';
END_PROGRAM

(* POU PDM_DISPLAY_SETTINGS/DISPLAY_SETTINGS, FBD *)
PROGRAM DISPLAY_SETTINGS
VAR


END_VAR

VAR_OUTPUT


END_VAR
VAR_INPUT
	INIT: BOOL;
END_VAR
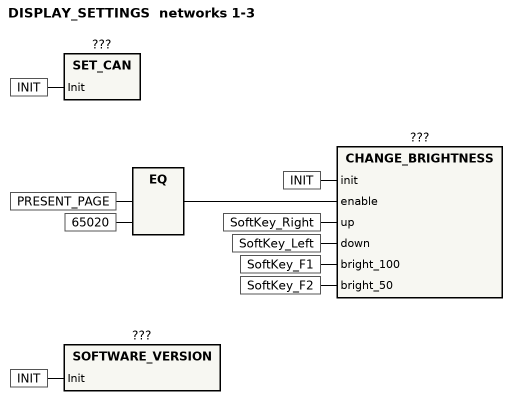
_FBD_ (* Function Block Diagram *)
NETWORK 1
	???:SET_CAN(Init: INIT)
NETWORK 2 (* Cange brightness *)
	???:CHANGE_BRIGHTNESS(init: INIT, enable: EQ(PRESENT_PAGE, 65020), up: SoftKey_Right, down: SoftKey_Left, bright_100: SoftKey_F1, bright_50: SoftKey_F2)
NETWORK 3
	???:SOFTWARE_VERSION(Init: INIT)
_END_FBD_
END_PROGRAM

(* POU PDM_DISPLAY_SETTINGS/SET_CAN, FBD *)
PROGRAM SET_CAN
VAR_INPUT
	Init: BOOL;
END_VAR
VAR
	SetLED: SET_LED;

	ResultLed: BYTE;
	SetLedStatus: BOOL:=TRUE;

	Color1: BYTE:=0;
	Color2: BYTE:=2;
	Frequency: BYTE:=2;
	CAN1: CAN_ENABLE;
	DesiredBaudrate: WORD;
	EnableBaudrate: BOOL;
	SetId: CAN_SETDOWNLOADID;
	Can1Status: CAN_STATUS;
	PresentDownloadId: BYTE;
	PresentBaudRate: WORD;
	Did: BYTE;
	DesiredDownloadId: BYTE;
	EnableDownloadId: BOOL;
	Waitstate: BOOL;
	ResultSeId: BYTE;
	PowerCyle: BOOL;
	TestInit: BOOL:=TRUE;

	ClearStatus: BOOL;
END_VAR
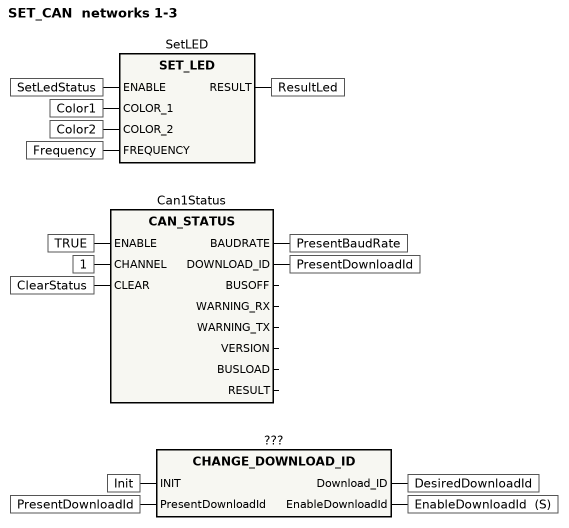
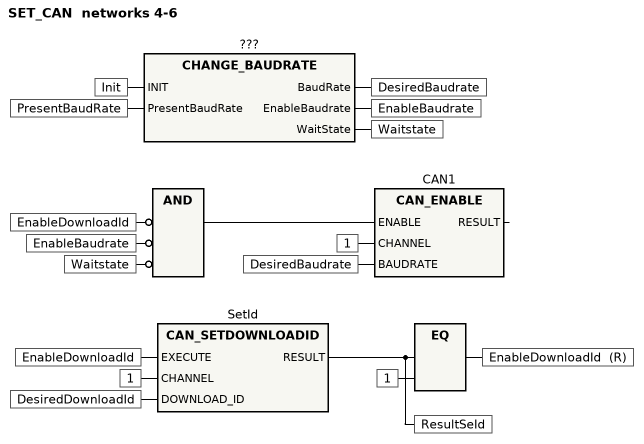
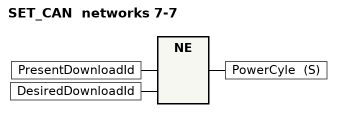
_FBD_ (* Function Block Diagram *)
NETWORK 1
	SetLED:SET_LED(ENABLE: SetLedStatus, COLOR_1: Color1, COLOR_2: Color2, FREQUENCY: Frequency) => ResultLed
NETWORK 2
	Can1Status:CAN_STATUS(ENABLE: TRUE, CHANNEL: 1, CLEAR: ClearStatus, DOWNLOAD_ID => PresentDownloadId) => PresentBaudRate
NETWORK 3
	???:CHANGE_DOWNLOAD_ID(INIT: Init, PresentDownloadId: PresentDownloadId, EnableDownloadId => S EnableDownloadId) => DesiredDownloadId
NETWORK 4
	???:CHANGE_BAUDRATE(INIT: Init, PresentBaudRate: PresentBaudRate, EnableBaudrate => EnableBaudrate, WaitState => Waitstate) => DesiredBaudrate
NETWORK 5
	CAN1:CAN_ENABLE(ENABLE: AND(NOT EnableDownloadId, NOT EnableBaudrate, NOT Waitstate), CHANNEL: 1, BAUDRATE: DesiredBaudrate)
NETWORK 6
	EQ(<SetId:CAN_SETDOWNLOADID(EXECUTE: EnableDownloadId, CHANNEL: 1, DOWNLOAD_ID: DesiredDownloadId) => ResultSeId>, 1) => R EnableDownloadId
NETWORK 7
	NE(PresentDownloadId, DesiredDownloadId) => S PowerCyle
_END_FBD_
(* the same logic as Structured Text *)
(* Network 1 *)
SetLED(ENABLE := SetLedStatus, COLOR_1 := Color1, COLOR_2 := Color2, FREQUENCY := Frequency);
ResultLed := SetLED.RESULT;
(* Network 2 *)
Can1Status(ENABLE := TRUE, CHANNEL := 1, CLEAR := ClearStatus);
PresentDownloadId := Can1Status.DOWNLOAD_ID;
PresentBaudRate := Can1Status.BAUDRATE;
(* Network 3: see the listing above *)
(* Network 4: see the listing above *)
(* Network 5 *)
CAN1(ENABLE := NOT EnableDownloadId AND NOT EnableBaudrate AND NOT Waitstate, CHANNEL := 1, BAUDRATE := DesiredBaudrate);
(* Network 6 *)
SetId(EXECUTE := EnableDownloadId, CHANNEL := 1, DOWNLOAD_ID := DesiredDownloadId);
ResultSeId := SetId.RESULT;
IF SetId.RESULT = 1 THEN EnableDownloadId := FALSE; END_IF;
(* Network 7 *)
IF PresentDownloadId <> DesiredDownloadId THEN PowerCyle := TRUE; END_IF;
END_PROGRAM

(* POU PDM_DISPLAY_SETTINGS/CHANGE_DOWNLOAD_ID, ST *)
PROGRAM CHANGE_DOWNLOAD_ID

VAR
	BaudArray: ARRAY[0..7] OF WORD := 10,20,50,125,250,500,800,1000;
	index: BYTE := 3;

	Id: BYTE;
	WaitState: BOOL;
	Download_IDIntern: BYTE;
END_VAR
VAR_INPUT
	INIT:BOOL;
	PresentDownloadId:BYTE;
END_VAR

VAR_OUTPUT
	Download_ID: BYTE;
	EnableDownloadId: BOOL;
END_VAR
	IF INIT THEN
		WaitState:=TRUE;
	END_IF;
	IF WaitState THEN
		IF PresentDownloadId<>0 THEN
			Download_ID:=PresentDownloadId;
			Id:=PresentDownloadId;
			WaitState:=FALSE;
		END_IF;
	END_IF;

	EnableDownloadId:=FALSE;

	IF PRESENT_PAGE = 65030 THEN
		IF SoftKey_Right AND NOT SoftKey2_F1 THEN
			Id:=Id+1;
		END_IF;
		IF SoftKey_Right AND SoftKey2_F1 THEN
			Id:=Id+10;
		END_IF;

		IF SoftKey_Left AND NOT SoftKey2_F1 THEN
			Id:=Id-1;
		END_IF;
		IF SoftKey_left AND SoftKey2_F1 THEN
			Id:=Id-10;
		END_IF;

		IF Id > 127 THEN
			Id:=127;
		END_IF;
		IF Id < 1 THEN
			Id:=1;
		END_IF;

		IF SoftKey_OK THEN
			EnableDownloadId:=SoftKey_OK;
			Download_ID:=Id;
		END_IF;
	END_IF;
END_PROGRAM

(* POU PDM_DISPLAY_SETTINGS/CHANGE_BAUDRATE, ST *)
PROGRAM CHANGE_BAUDRATE

VAR
	BaudArray: ARRAY[0..7] OF WORD := 10,20,50,125,250,500,800,1000;
	index: BYTE;

	BaudRateIntern: WORD;

END_VAR
VAR_INPUT
	INIT:BOOL;
	PresentBaudRate:WORD;
END_VAR
VAR_OUTPUT
	BaudRate:WORD;
	EnableBaudrate: BOOL;
	WaitState: BOOL;
END_VAR
	IF INIT THEN
		WaitState:=TRUE;
	END_IF;
	IF WaitState THEN
		IF PresentBaudRate<>0 THEN
			BaudRate:=PresentBaudRate;
			WaitState:=FALSE;
			CASE BaudRate OF
				10:
					Index:=0;
				20:
					Index:=1;
				50:
					Index:=2;
				125:
					Index:=3;
				250:
					Index:=4;
				500:
					Index:=5;
				800:
					Index:=6;
				1000:
					Index:=7;
			END_CASE;
		END_IF;
	END_IF;

	EnableBaudrate:=FALSE;

	IF PRESENT_PAGE = 65040 THEN
		IF SoftKey_Right THEN
			index:=Index+1;
		END_IF;
		IF SoftKey_Left THEN
			index:=Index-1;
		END_IF;
		IF index > 7 THEN
			index:=7;
		END_IF;

		BaudRateIntern:=BaudArray[index];
		IF SoftKey_OK THEN
			BaudRate:=BaudRateIntern;
			EnableBaudrate:=TRUE;
		END_IF;

	END_IF;
END_PROGRAM

(* POU PDM_DISPLAY_SETTINGS/CHANGE_BRIGHTNESS, ST *)
PROGRAM CHANGE_BRIGHTNESS
VAR_OUTPUT

END_VAR
VAR_INPUT

	init: BOOL;
	enable: BOOL;
	up: BOOL;
	down: BOOL;
	bright_100: BOOL;
	bright_50: BOOL;

END_VAR
VAR

	bright_old: BYTE;
	extern: BOOL;
	init2: BOOL;
	TON_Delay: TON;
END_VAR

VAR RETAIN
	bright_: BYTE;
END_VAR
(*Reload brightness BACKLIGHT is in the 2 cycle available*)

	IF  NOT init AND NOT init2 THEN
		IF bright_<1 THEN
			bright_:=100;
		ELSE
			SCREEN_BACKLIGHT_CTRL:=bright_;
		END_IF;
	END_IF;

	TON_Delay(IN:=Enable , PT:=T#100ms , Q=> , ET=> );

IF TON_Delay.Q THEN
(*incement/decrement brightness*)
	IF up THEN
		bright_:=bright_+1;
	END_IF;
	IF down  THEN
		bright_:=bright_-1;
	END_IF;
(*controll borders*)
	IF bright_<1 THEN
		bright_:=100;
	END_IF;
	IF bright_>100 OR bright_100 THEN
		bright_:=100;
	END_IF;
	IF  bright_50 THEN
		bright_:=50;
	END_IF;
END_IF;

(*if brightness settings come from outside e.g. from PLC*)
	IF bright_old<>DESIRED_BACKLIGHT THEN
		bright_old:=DESIRED_BACKLIGHT;
		extern:=TRUE;
	END_IF;

	IF DESIRED_BACKLIGHT>0 AND extern THEN
		bright_:=DESIRED_BACKLIGHT;
	END_IF;

	extern:=FALSE;

(*wait one cycle to write value to BACKLIGHT*)

	IF init2 THEN
		SCREEN_BACKLIGHT_CTRL:=bright_;
	END_IF;

	init2:=init;
END_PROGRAM

(* POU PDM_DISPLAY_SETTINGS/SOFTWARE_VERSION, ST *)
PROGRAM SOFTWARE_VERSION
VAR
	ApplicationName:STRING[40];
	OperatingSystem:STRING[40];
	OrderNumber : STRING[40];


	GET_HW_INFO1: GET_HW_INFO;
	GET_SW_INFO1: GET_SW_INFO;
	GET_APP_INFO1: GET_APP_INFO;
	SET_IDENTITY1: SET_IDENTITY;
	GET_IDENTITY1: GET_IDENTITY;
END_VAR
VAR_INPUT
	Init: BOOL;
END_VAR
	SET_IDENTITY1(ENABLE:=Init , APP_IDENT:='ifm_template_CR0451Master_V020000_VBeta1' , RESULT=> );


	GET_HW_INFO1(
	ENABLE:=Init ,
	ORDER_NUM=>OrderNumber ,
	NAME=> ,
	SERIAL=> , 
	REVISION=> , 
	MAN_DATE=> ,
	RESULT=> );

	GET_SW_INFO1(
	ENABLE:=Init ,
	NAME=> ,
	VERSION=>OperatingSystem ,
	BUILD_NUM=> ,
	BUILD_DATE=> ,
	RESULT=> );

	GET_APP_INFO1(
	ENABLE:=Init ,
	NAME=> ,
	VERSION=> ,
	BUILD_NUM=> ,
	BUILD_DATE=> ,
	RESULT=> );


	GET_IDENTITY1(ENABLE:=Init , APP_IDENT=>ApplicationName , RESULT=> );
END_PROGRAM

(* POU PLC_CYCLE, ST *)
PROGRAM PLC_CYCLE
VAR
	old_cycle: DWORD;
	TIMER_READ_US1: TIMER_READ_US;
	cycle: DWORD;
	init: BOOL:=TRUE;
END_VAR
VAR_OUTPUT
	cycletime_us: DWORD;
	max_cycle_us: DWORD;
END_VAR

VAR_INPUT
	reset_max_cycletime: BOOL;
END_VAR
	TIMER_READ_US1(TIME_US=>cycle );
	cycletime_us:=cycle-old_cycle;
	old_cycle:=cycle;

	IF max_cycle_us<cycletime_us AND NOT init THEN
		max_cycle_us:=cycletime_us;
	END_IF;

	IF reset_max_cycletime THEN
		max_cycle_us:=0;
	END_IF;

	init:=FALSE;
END_PROGRAM

(* Visualisation MasterLayout_1
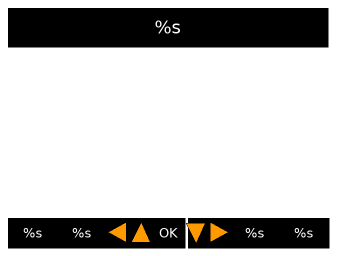
rectangle at (0,0)-(320,39): text "%s"; shows .TXT_HeadLine; invisible if .Hidden_HeadLine
rectangle at (271,210)-(321,240): text "%s"; shows .TXT_F4; invisible if .Hidden_F4
rectangle at (49,210)-(99,240): text "%s"; shows .TXT_F2; invisible if .Hidden_F2
rectangle at (0,210)-(50,240): text "%s"; shows .TXT_F1; invisible if .Hidden_F1
rectangle at (98,210)-(122,240): invisible if .Hidden_Left
rectangle at (222,210)-(272,240): text "%s"; shows .TXT_F3; invisible if .Hidden_F3
polygon at (100,214)-(118,234): invisible if .Hidden_Left
rectangle at (144,210)-(177,240): text "OK"; invisible if .Hidden_Ok
rectangle at (121,210)-(145,240): invisible if .Hidden_Up
rectangle at (180,210)-(204,240): invisible if .Hidden_Down
rectangle at (199,210)-(223,240): invisible if .Hidden_Right
polygon at (202,214)-(220,234): invisible if .Hidden_Right
polygon at (123,214)-(142,234): invisible if .Hidden_Up
polygon at (178,215)-(197,235): invisible if .Hidden_Down
*)

(* Visualisation START_PAGE/P00001
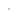
bitmap at (0,0)-(1,1): c:\users\oliver\downloads\mm_blank_320x240RLE.bmp
*)

(* Visualisation START_PAGE/MAIN_MANU/MAIN_MENU_1/P00010
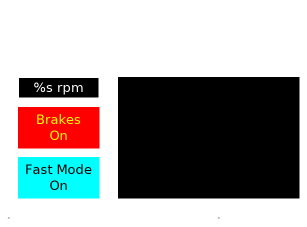
bitmap at (10,210)-(11,211): c:\users\oliver\downloads\settings+icon-1320184981403058053RLE.bmp
rectangle at (20,0)-(301,41): text "SKYLINE OFF"
bitmap at (220,210)-(221,211): j:\research and development\r&d department (inprogress)\2 - projects\32900 modern machinery hydraulic skyline control\2 - development stage\graphics\off_toggleRLE.bmp
rectangle at (120,70)-(211,131): text "WARNING! / Overload"; invisible if NOT.overloadWarningBlink
rectangle at (120,130)-(211,191): text "WARNING! / Sensor Fail"; invisible if NOT.sensorFailureBlink
rectangle at (210,70)-(301,131): text "WARNING! / Overspeed"; invisible if NOT.overspeedAlarmBlink
rectangle at (210,130)-(301,191): text "CAUTION! / Slow Down"; invisible if NOT.overspeedWarning
rectangle at (20,70)-(101,91): text "%s rpm"; shows REAL_TO_INT((encoderHz*60*34.2)/500)
rectangle at (120,40)-(301,71): text "Alarms grid:"
rectangle at (20,40)-(101,71): text "Speed:"
rectangle at (20,100)-(101,141): text "Brakes / Off"; invisible if brakesOn
rectangle at (20,150)-(101,191): text "Fast Mode / Off"; invisible if highSpeedMode
rectangle at (20,100)-(101,141): text "Brakes / On"; invisible if NOT.brakesAlarm
rectangle at (20,150)-(101,191): text "Fast Mode / On"; invisible if NOT.highSpeedMode
4 more shapes without text or variables
*)

(* Visualisation START_PAGE/MAIN_MANU/MAIN_MENU_1/P00011
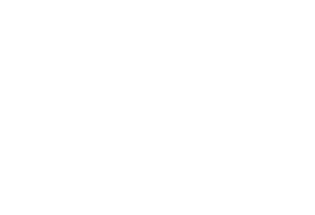
rectangle at (20,40)-(221,71): text "Encoder pulse count :"
rectangle at (230,40)-(301,71): text "%s"; shows encoderCount
rectangle at (230,70)-(301,101): text "%s"; shows motorWindinPsi
rectangle at (270,210)-(321,241): text "ESC"
rectangle at (270,210)-(321,241): text "ESC"; invisible if NOT.alarm
rectangle at (20,70)-(221,101): text "Motor port A psi :"
rectangle at (20,100)-(221,131): text "Motor port B psi :"
rectangle at (230,100)-(311,131): text "%s"; shows motorPayoutPsi
rectangle at (20,130)-(231,161): text "Joystick input :"
rectangle at (230,130)-(301,161): text "%s V"; shows joystick/1000
rectangle at (20,160)-(231,191): text "Fast mode button :"
rectangle at (230,160)-(301,191): text "%s"; shows boostButton
*)

(* Visualisation START_PAGE/MAIN_MANU/MAIN_MENU_1/P00012
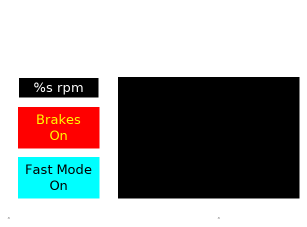
rectangle at (20,100)-(101,141): text "Brakes / Off"; invisible if brakesOn
rectangle at (20,150)-(101,191): text "Fast Mode / Off"; invisible if highSpeedMode
rectangle at (20,0)-(301,41): text "SKYLINE ON"
rectangle at (120,70)-(211,131): text "WARNING! / Overload"; invisible if NOT.overloadWarningBlink
rectangle at (120,130)-(211,191): text "WARNING! / Sensor Fail"; invisible if NOT.sensorFailureBlink
bitmap at (10,210)-(11,211): c:\users\oliver\downloads\settings+icon-1320184981403058053RLE.bmp
bitmap at (220,210)-(221,211): j:\research and development\r&d department (inprogress)\2 - projects\32900 modern machinery hydraulic skyline control\2 - development stage\graphics\on_toggleRLE.bmp
rectangle at (210,70)-(301,131): text "WARNING! / Overspeed"; invisible if NOT.overspeedAlarmBlink
rectangle at (210,130)-(301,191): text "CAUTION! / Slow Down"; invisible if NOT.overspeedWarning
rectangle at (20,70)-(101,91): text "%s rpm"; shows REAL_TO_INT((encoderHz*60*34.2)/500)
rectangle at (120,40)-(301,71): text "Alarms grid:"
rectangle at (20,40)-(101,71): text "Speed:"
rectangle at (20,100)-(101,141): text "Brakes / On"; invisible if NOT.brakesAlarm
rectangle at (20,150)-(101,191): text "Fast Mode / On"; invisible if NOT.highSpeedMode
4 more shapes without text or variables
*)

(* Visualisation START_PAGE/MAIN_MANU/MAIN_MENU_1/P00013
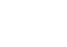
rectangle at (270,210)-(321,241): text "ESC"
rectangle at (270,210)-(321,241): text "ESC"; invisible if NOT.alarm
*)

(* Visualisation START_PAGE/MAIN_MANU/MAIN_MENU_1/P00014
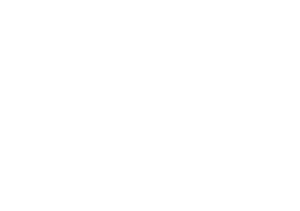
rectangle at (110,40)-(291,71): text "%s"; shows CONCAT(prefix, cr0403VersionNo)
rectangle at (110,70)-(291,101): text "%s"; shows CONCAT(prefix, cr0431VersionNo)
rectangle at (110,100)-(291,131): text "%s"; shows CONCAT(prefix, cr0451VersionNo)
rectangle at (20,40)-(111,71): text "CR0403:"
rectangle at (20,70)-(111,101): text "CR0431:"
rectangle at (20,100)-(111,131): text "CR0451:"
rectangle at (270,210)-(321,241): text "ESC"
rectangle at (270,210)-(321,241): text "ESC"; invisible if NOT.alarm
*)

(* Visualisation START_PAGE/MAIN_MANU/MAIN_MENU_1/P00015
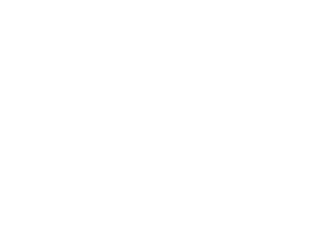
rectangle at (20,30)-(221,61): text "Motor swash output :"
rectangle at (230,30)-(301,61): text "%s %%"; shows motorSwash / 10
rectangle at (20,60)-(221,91): text "Water brake applied :"
rectangle at (20,90)-(221,121): text "Band brake applied :"
rectangle at (230,60)-(301,91): text "%s %%"; shows 100- (waterBrake / 10)
rectangle at (230,90)-(301,121): text "%s %%"; shows 100-(bandBrake / 10)
rectangle at (20,120)-(221,151): text "Warning buzzer :"
rectangle at (230,120)-(301,151): text "%s"; shows alarm
rectangle at (20,150)-(221,181): text "Skyline drum clutch :"
rectangle at (20,180)-(221,211): text "Park brake :"
rectangle at (270,210)-(321,241): text "ESC"
rectangle at (270,210)-(321,241): text "ESC"; invisible if NOT.alarm
rectangle at (230,150)-(301,181): text "%s"; shows skylineClutch
rectangle at (230,180)-(301,211): text "%s"; shows parkBrake
*)

(* Visualisation START_PAGE/MAIN_MANU/MAIN_MENU_1/P00016
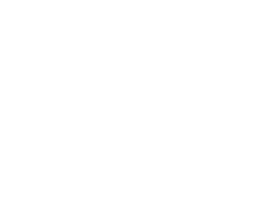
rectangle at (20,70)-(302,101): text "Input Status"; alarm colour if SELECT_PAGE.MenuItem=2
rectangle at (20,40)-(302,71): text "Setpoints"; alarm colour if SELECT_PAGE.MenuItem=1
rectangle at (20,100)-(302,131): text "Output Status"; alarm colour if SELECT_PAGE.MenuItem=3
rectangle at (20,130)-(302,161): text "Alarms Log"; alarm colour if SELECT_PAGE.MenuItem=4
rectangle at (270,210)-(321,241): text "ESC"
rectangle at (270,210)-(321,241): text "ESC"
rectangle at (270,210)-(321,241): text "ESC"; invisible if NOT.alarm
rectangle at (20,160)-(302,191): text "Software Version"; alarm colour if SELECT_PAGE.MenuItem=5
*)

(* Visualisation START_PAGE/MAIN_MANU/MAIN_MENU_1/DISPLAY_SETUP/1_DISPLAY_SETUP/1_Set_Band_Brake_Limit/P60013
